// TIA Portal V17 export
// export: Created 2025-07-01T09:58:33.5756793Z, ExportSetting WithDefaults, DisplayName Totally Integrated Automation Portal, DisplayVersion V17 Update 8, DisplayName TIA Portal Openness, DisplayVersion V17 Update 8, DisplayName TIA Portal Version Control Interface, DisplayVersion V17, DisplayName SINAMICS Startdrive Advanced, DisplayVersion V17 SP2, DisplayName SINAMICS Startdrive G110M, G120, G120C, G120D, G120P, G115D, DisplayVersion V17 SP2, DisplayName SINAMICS Startdrive G130, G150, S120, S150, SINAMICS MV, S210, DisplayVersion V17 SP2, DisplayName STEP 7 Professional, DisplayVersion V17 Update 8, DisplayName SINUMERIK ONE STEP 7 Toolbox, DisplayVersion V17 Update 12, DisplayName SINUMERIK ONE PLC Basic Program Plus, DisplayVersion V17 Update 12, DisplayName SINUMERIK 840D sl STEP 7 Toolbox, DisplayVersion V17 Update 12, DisplayName STEP 7 Safety, DisplayVersion V17 Update 6, DisplayName WinCC Advanced, DisplayVersion V17 Update 8
FUNCTION "FC349_NCK_M_CH2_UNIT_1_STA_3" : Void   // FC349, LAD
TITLE = Channel 1 data
{ S7_Optimized_Access := 'FALSE' }
AUTHOR : ETXETAR
VERSION : 1.0
// stored: AutoNumber false, IsIECCheckEnabled false, SetENOAutomatically false, UDAEnableTagReadback false
BEGIN

REGION Network 1: ACKNOWLEDGE M704-FIXTURE 4 VERIFY PART AND TOOL IS CLAMPED DURING MACHINING (WHEN TRUE DO). TOGGLED / ACKNOWLEDGE M46-VERIFY FIXTURE 1 PART AND TOOL IS CLAMPED DURING
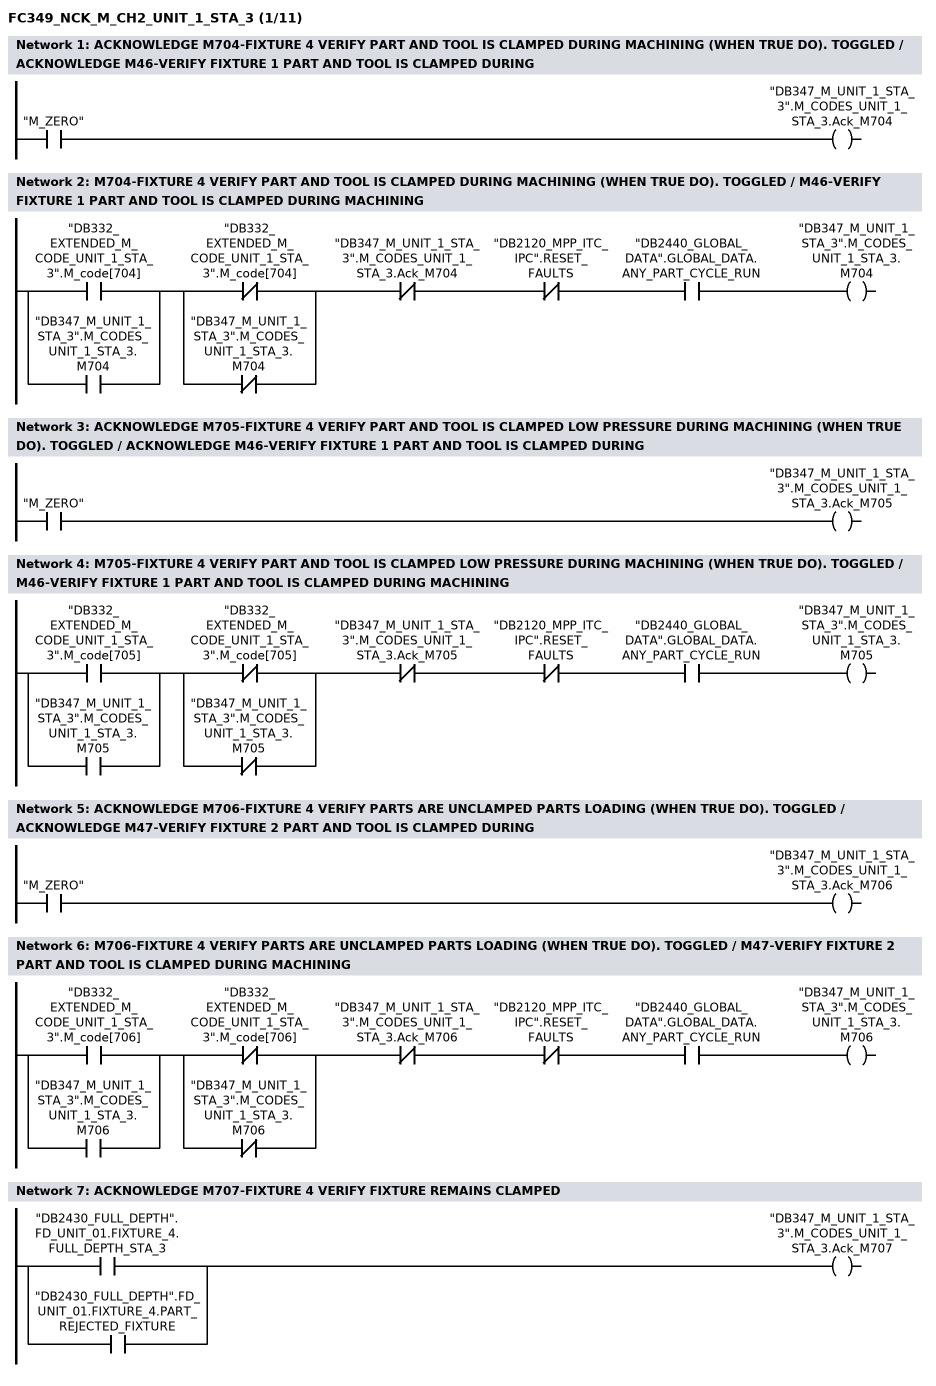
   RUNG wire#powerrail
      Contact( "M_ZERO" )
      Coil( "DB347_M_UNIT_1_STA_3".M_CODES_UNIT_1_STA_3.Ack_M704 )
   END_RUNG
   // the same network as SCL:
   "DB347_M_UNIT_1_STA_3".M_CODES_UNIT_1_STA_3.Ack_M704 := "M_ZERO";
END_REGION

REGION Network 2: M704-FIXTURE 4 VERIFY PART AND TOOL IS CLAMPED DURING MACHINING (WHEN TRUE DO). TOGGLED / M46-VERIFY FIXTURE 1 PART AND TOOL IS CLAMPED DURING MACHINING
   RUNG wire#powerrail
      Contact( "DB332_EXTENDED_M_CODE_UNIT_1_STA_3".M_code[704] )
      wire#w1
      I_Contact( "DB332_EXTENDED_M_CODE_UNIT_1_STA_3".M_code[704] )
      wire#w2
      I_Contact( "DB347_M_UNIT_1_STA_3".M_CODES_UNIT_1_STA_3.Ack_M704 )
      I_Contact( "DB2120_MPP_ITC_IPC".RESET_FAULTS )
      Contact( "DB2440_GLOBAL_DATA".GLOBAL_DATA.ANY_PART_CYCLE_RUN )
      Coil( "DB347_M_UNIT_1_STA_3".M_CODES_UNIT_1_STA_3.M704 )
   END_RUNG
   RUNG wire#powerrail
      Contact( "DB347_M_UNIT_1_STA_3".M_CODES_UNIT_1_STA_3.M704 )
   END_RUNG wire#w1
   RUNG wire#w1
      I_Contact( "DB347_M_UNIT_1_STA_3".M_CODES_UNIT_1_STA_3.M704 )
   END_RUNG wire#w2
   // the same network as SCL:
   "DB347_M_UNIT_1_STA_3".M_CODES_UNIT_1_STA_3.M704 := ("DB332_EXTENDED_M_CODE_UNIT_1_STA_3".M_code[704] OR "DB347_M_UNIT_1_STA_3".M_CODES_UNIT_1_STA_3.M704) AND (NOT "DB332_EXTENDED_M_CODE_UNIT_1_STA_3".M_code[704] OR NOT "DB347_M_UNIT_1_STA_3".M_CODES_UNIT_1_STA_3.M704) AND NOT "DB347_M_UNIT_1_STA_3".M_CODES_UNIT_1_STA_3.Ack_M704 AND NOT "DB2120_MPP_ITC_IPC".RESET_FAULTS AND "DB2440_GLOBAL_DATA".GLOBAL_DATA.ANY_PART_CYCLE_RUN;
END_REGION

REGION Network 3: ACKNOWLEDGE M705-FIXTURE 4 VERIFY PART AND TOOL IS CLAMPED LOW PRESSURE DURING MACHINING (WHEN TRUE DO). TOGGLED / ACKNOWLEDGE M46-VERIFY FIXTURE 1 PART AND TOOL IS CLAMPED DURING
   RUNG wire#powerrail
      Contact( "M_ZERO" )
      Coil( "DB347_M_UNIT_1_STA_3".M_CODES_UNIT_1_STA_3.Ack_M705 )
   END_RUNG
   // the same network as SCL:
   "DB347_M_UNIT_1_STA_3".M_CODES_UNIT_1_STA_3.Ack_M705 := "M_ZERO";
END_REGION

REGION Network 4: M705-FIXTURE 4 VERIFY PART AND TOOL IS CLAMPED LOW PRESSURE DURING MACHINING (WHEN TRUE DO). TOGGLED / M46-VERIFY FIXTURE 1 PART AND TOOL IS CLAMPED DURING MACHINING
   RUNG wire#powerrail
      Contact( "DB332_EXTENDED_M_CODE_UNIT_1_STA_3".M_code[705] )
      wire#w1
      I_Contact( "DB332_EXTENDED_M_CODE_UNIT_1_STA_3".M_code[705] )
      wire#w2
      I_Contact( "DB347_M_UNIT_1_STA_3".M_CODES_UNIT_1_STA_3.Ack_M705 )
      I_Contact( "DB2120_MPP_ITC_IPC".RESET_FAULTS )
      Contact( "DB2440_GLOBAL_DATA".GLOBAL_DATA.ANY_PART_CYCLE_RUN )
      Coil( "DB347_M_UNIT_1_STA_3".M_CODES_UNIT_1_STA_3.M705 )
   END_RUNG
   RUNG wire#powerrail
      Contact( "DB347_M_UNIT_1_STA_3".M_CODES_UNIT_1_STA_3.M705 )
   END_RUNG wire#w1
   RUNG wire#w1
      I_Contact( "DB347_M_UNIT_1_STA_3".M_CODES_UNIT_1_STA_3.M705 )
   END_RUNG wire#w2
   // the same network as SCL:
   "DB347_M_UNIT_1_STA_3".M_CODES_UNIT_1_STA_3.M705 := ("DB332_EXTENDED_M_CODE_UNIT_1_STA_3".M_code[705] OR "DB347_M_UNIT_1_STA_3".M_CODES_UNIT_1_STA_3.M705) AND (NOT "DB332_EXTENDED_M_CODE_UNIT_1_STA_3".M_code[705] OR NOT "DB347_M_UNIT_1_STA_3".M_CODES_UNIT_1_STA_3.M705) AND NOT "DB347_M_UNIT_1_STA_3".M_CODES_UNIT_1_STA_3.Ack_M705 AND NOT "DB2120_MPP_ITC_IPC".RESET_FAULTS AND "DB2440_GLOBAL_DATA".GLOBAL_DATA.ANY_PART_CYCLE_RUN;
END_REGION

REGION Network 5: ACKNOWLEDGE M706-FIXTURE 4 VERIFY PARTS ARE UNCLAMPED PARTS LOADING (WHEN TRUE DO). TOGGLED / ACKNOWLEDGE M47-VERIFY FIXTURE 2 PART AND TOOL IS CLAMPED DURING
   RUNG wire#powerrail
      Contact( "M_ZERO" )
      Coil( "DB347_M_UNIT_1_STA_3".M_CODES_UNIT_1_STA_3.Ack_M706 )
   END_RUNG
   // the same network as SCL:
   "DB347_M_UNIT_1_STA_3".M_CODES_UNIT_1_STA_3.Ack_M706 := "M_ZERO";
END_REGION

REGION Network 6: M706-FIXTURE 4 VERIFY PARTS ARE UNCLAMPED PARTS LOADING (WHEN TRUE DO). TOGGLED / M47-VERIFY FIXTURE 2 PART AND TOOL IS CLAMPED DURING MACHINING
   RUNG wire#powerrail
      Contact( "DB332_EXTENDED_M_CODE_UNIT_1_STA_3".M_code[706] )
      wire#w1
      I_Contact( "DB332_EXTENDED_M_CODE_UNIT_1_STA_3".M_code[706] )
      wire#w2
      I_Contact( "DB347_M_UNIT_1_STA_3".M_CODES_UNIT_1_STA_3.Ack_M706 )
      I_Contact( "DB2120_MPP_ITC_IPC".RESET_FAULTS )
      Contact( "DB2440_GLOBAL_DATA".GLOBAL_DATA.ANY_PART_CYCLE_RUN )
      Coil( "DB347_M_UNIT_1_STA_3".M_CODES_UNIT_1_STA_3.M706 )
   END_RUNG
   RUNG wire#powerrail
      Contact( "DB347_M_UNIT_1_STA_3".M_CODES_UNIT_1_STA_3.M706 )
   END_RUNG wire#w1
   RUNG wire#w1
      I_Contact( "DB347_M_UNIT_1_STA_3".M_CODES_UNIT_1_STA_3.M706 )
   END_RUNG wire#w2
   // the same network as SCL:
   "DB347_M_UNIT_1_STA_3".M_CODES_UNIT_1_STA_3.M706 := ("DB332_EXTENDED_M_CODE_UNIT_1_STA_3".M_code[706] OR "DB347_M_UNIT_1_STA_3".M_CODES_UNIT_1_STA_3.M706) AND (NOT "DB332_EXTENDED_M_CODE_UNIT_1_STA_3".M_code[706] OR NOT "DB347_M_UNIT_1_STA_3".M_CODES_UNIT_1_STA_3.M706) AND NOT "DB347_M_UNIT_1_STA_3".M_CODES_UNIT_1_STA_3.Ack_M706 AND NOT "DB2120_MPP_ITC_IPC".RESET_FAULTS AND "DB2440_GLOBAL_DATA".GLOBAL_DATA.ANY_PART_CYCLE_RUN;
END_REGION

REGION Network 7: ACKNOWLEDGE M707-FIXTURE 4 VERIFY FIXTURE REMAINS CLAMPED
   RUNG wire#powerrail
      Contact( "DB2430_FULL_DEPTH".FD_UNIT_01.FIXTURE_4.FULL_DEPTH_STA_3 )
      wire#w1
      Coil( "DB347_M_UNIT_1_STA_3".M_CODES_UNIT_1_STA_3.Ack_M707 )
   END_RUNG
   RUNG wire#powerrail
      Contact( "DB2430_FULL_DEPTH".FD_UNIT_01.FIXTURE_4.PART_REJECTED_FIXTURE )
   END_RUNG wire#w1
   // the same network as SCL:
   "DB347_M_UNIT_1_STA_3".M_CODES_UNIT_1_STA_3.Ack_M707 := "DB2430_FULL_DEPTH".FD_UNIT_01.FIXTURE_4.FULL_DEPTH_STA_3 OR "DB2430_FULL_DEPTH".FD_UNIT_01.FIXTURE_4.PART_REJECTED_FIXTURE;
END_REGION

REGION Network 8: M707-FIXTURE 4 VERIFY FIXTURE REMAINS CLAMPED
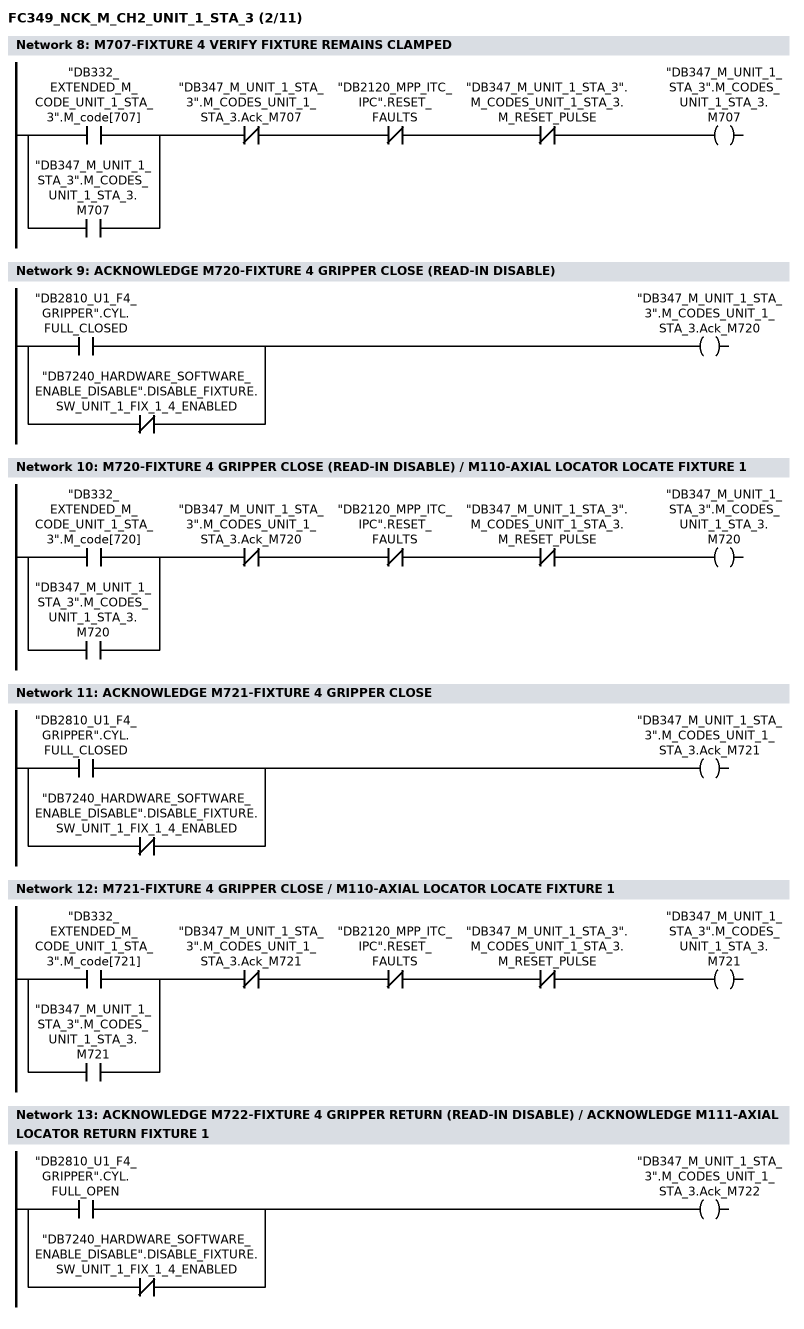
   RUNG wire#powerrail
      Contact( "DB332_EXTENDED_M_CODE_UNIT_1_STA_3".M_code[707] )
      wire#w1
      I_Contact( "DB347_M_UNIT_1_STA_3".M_CODES_UNIT_1_STA_3.Ack_M707 )
      I_Contact( "DB2120_MPP_ITC_IPC".RESET_FAULTS )
      I_Contact( "DB347_M_UNIT_1_STA_3".M_CODES_UNIT_1_STA_3.M_RESET_PULSE )
      Coil( "DB347_M_UNIT_1_STA_3".M_CODES_UNIT_1_STA_3.M707 )
   END_RUNG
   RUNG wire#powerrail
      Contact( "DB347_M_UNIT_1_STA_3".M_CODES_UNIT_1_STA_3.M707 )
   END_RUNG wire#w1
   // the same network as SCL:
   "DB347_M_UNIT_1_STA_3".M_CODES_UNIT_1_STA_3.M707 := ("DB332_EXTENDED_M_CODE_UNIT_1_STA_3".M_code[707] OR "DB347_M_UNIT_1_STA_3".M_CODES_UNIT_1_STA_3.M707) AND NOT "DB347_M_UNIT_1_STA_3".M_CODES_UNIT_1_STA_3.Ack_M707 AND NOT "DB2120_MPP_ITC_IPC".RESET_FAULTS AND NOT "DB347_M_UNIT_1_STA_3".M_CODES_UNIT_1_STA_3.M_RESET_PULSE;
END_REGION

REGION Network 9: ACKNOWLEDGE M720-FIXTURE 4 GRIPPER CLOSE (READ-IN DISABLE)
   RUNG wire#powerrail
      Contact( "DB2810_U1_F4_GRIPPER".CYL.FULL_CLOSED )
      wire#w1
      Coil( "DB347_M_UNIT_1_STA_3".M_CODES_UNIT_1_STA_3.Ack_M720 )
   END_RUNG
   RUNG wire#powerrail
      I_Contact( "DB7240_HARDWARE_SOFTWARE_ENABLE_DISABLE".DISABLE_FIXTURE.SW_UNIT_1_FIX_1_4_ENABLED )
   END_RUNG wire#w1
   // the same network as SCL:
   "DB347_M_UNIT_1_STA_3".M_CODES_UNIT_1_STA_3.Ack_M720 := "DB2810_U1_F4_GRIPPER".CYL.FULL_CLOSED OR NOT "DB7240_HARDWARE_SOFTWARE_ENABLE_DISABLE".DISABLE_FIXTURE.SW_UNIT_1_FIX_1_4_ENABLED;
END_REGION

REGION Network 10: M720-FIXTURE 4 GRIPPER CLOSE (READ-IN DISABLE) / M110-AXIAL LOCATOR LOCATE FIXTURE 1
   RUNG wire#powerrail
      Contact( "DB332_EXTENDED_M_CODE_UNIT_1_STA_3".M_code[720] )
      wire#w1
      I_Contact( "DB347_M_UNIT_1_STA_3".M_CODES_UNIT_1_STA_3.Ack_M720 )
      I_Contact( "DB2120_MPP_ITC_IPC".RESET_FAULTS )
      I_Contact( "DB347_M_UNIT_1_STA_3".M_CODES_UNIT_1_STA_3.M_RESET_PULSE )
      Coil( "DB347_M_UNIT_1_STA_3".M_CODES_UNIT_1_STA_3.M720 )
   END_RUNG
   RUNG wire#powerrail
      Contact( "DB347_M_UNIT_1_STA_3".M_CODES_UNIT_1_STA_3.M720 )
   END_RUNG wire#w1
   // the same network as SCL:
   "DB347_M_UNIT_1_STA_3".M_CODES_UNIT_1_STA_3.M720 := ("DB332_EXTENDED_M_CODE_UNIT_1_STA_3".M_code[720] OR "DB347_M_UNIT_1_STA_3".M_CODES_UNIT_1_STA_3.M720) AND NOT "DB347_M_UNIT_1_STA_3".M_CODES_UNIT_1_STA_3.Ack_M720 AND NOT "DB2120_MPP_ITC_IPC".RESET_FAULTS AND NOT "DB347_M_UNIT_1_STA_3".M_CODES_UNIT_1_STA_3.M_RESET_PULSE;
END_REGION

REGION Network 11: ACKNOWLEDGE M721-FIXTURE 4 GRIPPER CLOSE
   RUNG wire#powerrail
      Contact( "DB2810_U1_F4_GRIPPER".CYL.FULL_CLOSED )
      wire#w1
      Coil( "DB347_M_UNIT_1_STA_3".M_CODES_UNIT_1_STA_3.Ack_M721 )
   END_RUNG
   RUNG wire#powerrail
      I_Contact( "DB7240_HARDWARE_SOFTWARE_ENABLE_DISABLE".DISABLE_FIXTURE.SW_UNIT_1_FIX_1_4_ENABLED )
   END_RUNG wire#w1
   // the same network as SCL:
   "DB347_M_UNIT_1_STA_3".M_CODES_UNIT_1_STA_3.Ack_M721 := "DB2810_U1_F4_GRIPPER".CYL.FULL_CLOSED OR NOT "DB7240_HARDWARE_SOFTWARE_ENABLE_DISABLE".DISABLE_FIXTURE.SW_UNIT_1_FIX_1_4_ENABLED;
END_REGION

REGION Network 12: M721-FIXTURE 4 GRIPPER CLOSE / M110-AXIAL LOCATOR LOCATE FIXTURE 1
   RUNG wire#powerrail
      Contact( "DB332_EXTENDED_M_CODE_UNIT_1_STA_3".M_code[721] )
      wire#w1
      I_Contact( "DB347_M_UNIT_1_STA_3".M_CODES_UNIT_1_STA_3.Ack_M721 )
      I_Contact( "DB2120_MPP_ITC_IPC".RESET_FAULTS )
      I_Contact( "DB347_M_UNIT_1_STA_3".M_CODES_UNIT_1_STA_3.M_RESET_PULSE )
      Coil( "DB347_M_UNIT_1_STA_3".M_CODES_UNIT_1_STA_3.M721 )
   END_RUNG
   RUNG wire#powerrail
      Contact( "DB347_M_UNIT_1_STA_3".M_CODES_UNIT_1_STA_3.M721 )
   END_RUNG wire#w1
   // the same network as SCL:
   "DB347_M_UNIT_1_STA_3".M_CODES_UNIT_1_STA_3.M721 := ("DB332_EXTENDED_M_CODE_UNIT_1_STA_3".M_code[721] OR "DB347_M_UNIT_1_STA_3".M_CODES_UNIT_1_STA_3.M721) AND NOT "DB347_M_UNIT_1_STA_3".M_CODES_UNIT_1_STA_3.Ack_M721 AND NOT "DB2120_MPP_ITC_IPC".RESET_FAULTS AND NOT "DB347_M_UNIT_1_STA_3".M_CODES_UNIT_1_STA_3.M_RESET_PULSE;
END_REGION

REGION Network 13: ACKNOWLEDGE M722-FIXTURE 4 GRIPPER RETURN (READ-IN DISABLE) / ACKNOWLEDGE M111-AXIAL LOCATOR RETURN FIXTURE 1
   RUNG wire#powerrail
      Contact( "DB2810_U1_F4_GRIPPER".CYL.FULL_OPEN )
      wire#w1
      Coil( "DB347_M_UNIT_1_STA_3".M_CODES_UNIT_1_STA_3.Ack_M722 )
   END_RUNG
   RUNG wire#powerrail
      I_Contact( "DB7240_HARDWARE_SOFTWARE_ENABLE_DISABLE".DISABLE_FIXTURE.SW_UNIT_1_FIX_1_4_ENABLED )
   END_RUNG wire#w1
   // the same network as SCL:
   "DB347_M_UNIT_1_STA_3".M_CODES_UNIT_1_STA_3.Ack_M722 := "DB2810_U1_F4_GRIPPER".CYL.FULL_OPEN OR NOT "DB7240_HARDWARE_SOFTWARE_ENABLE_DISABLE".DISABLE_FIXTURE.SW_UNIT_1_FIX_1_4_ENABLED;
END_REGION

REGION Network 14: M722-FIXTURE 4 GRIPPER RETURN (READ-IN DISABLE) / M111-AXIAL LOCATOR RETURN FIXTURE 1
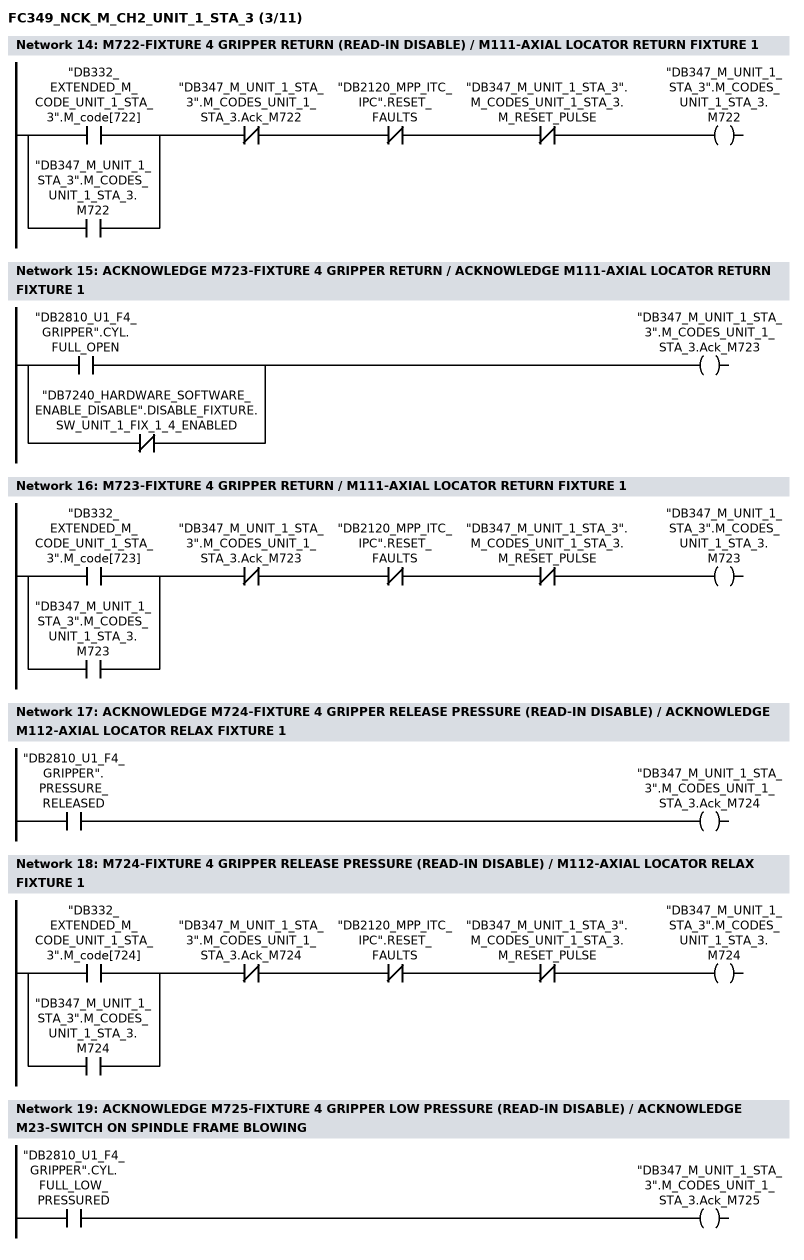
   RUNG wire#powerrail
      Contact( "DB332_EXTENDED_M_CODE_UNIT_1_STA_3".M_code[722] )
      wire#w1
      I_Contact( "DB347_M_UNIT_1_STA_3".M_CODES_UNIT_1_STA_3.Ack_M722 )
      I_Contact( "DB2120_MPP_ITC_IPC".RESET_FAULTS )
      I_Contact( "DB347_M_UNIT_1_STA_3".M_CODES_UNIT_1_STA_3.M_RESET_PULSE )
      Coil( "DB347_M_UNIT_1_STA_3".M_CODES_UNIT_1_STA_3.M722 )
   END_RUNG
   RUNG wire#powerrail
      Contact( "DB347_M_UNIT_1_STA_3".M_CODES_UNIT_1_STA_3.M722 )
   END_RUNG wire#w1
   // the same network as SCL:
   "DB347_M_UNIT_1_STA_3".M_CODES_UNIT_1_STA_3.M722 := ("DB332_EXTENDED_M_CODE_UNIT_1_STA_3".M_code[722] OR "DB347_M_UNIT_1_STA_3".M_CODES_UNIT_1_STA_3.M722) AND NOT "DB347_M_UNIT_1_STA_3".M_CODES_UNIT_1_STA_3.Ack_M722 AND NOT "DB2120_MPP_ITC_IPC".RESET_FAULTS AND NOT "DB347_M_UNIT_1_STA_3".M_CODES_UNIT_1_STA_3.M_RESET_PULSE;
END_REGION

REGION Network 15: ACKNOWLEDGE M723-FIXTURE 4 GRIPPER RETURN / ACKNOWLEDGE M111-AXIAL LOCATOR RETURN FIXTURE 1
   RUNG wire#powerrail
      Contact( "DB2810_U1_F4_GRIPPER".CYL.FULL_OPEN )
      wire#w1
      Coil( "DB347_M_UNIT_1_STA_3".M_CODES_UNIT_1_STA_3.Ack_M723 )
   END_RUNG
   RUNG wire#powerrail
      I_Contact( "DB7240_HARDWARE_SOFTWARE_ENABLE_DISABLE".DISABLE_FIXTURE.SW_UNIT_1_FIX_1_4_ENABLED )
   END_RUNG wire#w1
   // the same network as SCL:
   "DB347_M_UNIT_1_STA_3".M_CODES_UNIT_1_STA_3.Ack_M723 := "DB2810_U1_F4_GRIPPER".CYL.FULL_OPEN OR NOT "DB7240_HARDWARE_SOFTWARE_ENABLE_DISABLE".DISABLE_FIXTURE.SW_UNIT_1_FIX_1_4_ENABLED;
END_REGION

REGION Network 16: M723-FIXTURE 4 GRIPPER RETURN / M111-AXIAL LOCATOR RETURN FIXTURE 1
   RUNG wire#powerrail
      Contact( "DB332_EXTENDED_M_CODE_UNIT_1_STA_3".M_code[723] )
      wire#w1
      I_Contact( "DB347_M_UNIT_1_STA_3".M_CODES_UNIT_1_STA_3.Ack_M723 )
      I_Contact( "DB2120_MPP_ITC_IPC".RESET_FAULTS )
      I_Contact( "DB347_M_UNIT_1_STA_3".M_CODES_UNIT_1_STA_3.M_RESET_PULSE )
      Coil( "DB347_M_UNIT_1_STA_3".M_CODES_UNIT_1_STA_3.M723 )
   END_RUNG
   RUNG wire#powerrail
      Contact( "DB347_M_UNIT_1_STA_3".M_CODES_UNIT_1_STA_3.M723 )
   END_RUNG wire#w1
   // the same network as SCL:
   "DB347_M_UNIT_1_STA_3".M_CODES_UNIT_1_STA_3.M723 := ("DB332_EXTENDED_M_CODE_UNIT_1_STA_3".M_code[723] OR "DB347_M_UNIT_1_STA_3".M_CODES_UNIT_1_STA_3.M723) AND NOT "DB347_M_UNIT_1_STA_3".M_CODES_UNIT_1_STA_3.Ack_M723 AND NOT "DB2120_MPP_ITC_IPC".RESET_FAULTS AND NOT "DB347_M_UNIT_1_STA_3".M_CODES_UNIT_1_STA_3.M_RESET_PULSE;
END_REGION

REGION Network 17: ACKNOWLEDGE M724-FIXTURE 4 GRIPPER RELEASE PRESSURE (READ-IN DISABLE) / ACKNOWLEDGE M112-AXIAL LOCATOR RELAX FIXTURE 1
   RUNG wire#powerrail
      Contact( "DB2810_U1_F4_GRIPPER".PRESSURE_RELEASED )
      Coil( "DB347_M_UNIT_1_STA_3".M_CODES_UNIT_1_STA_3.Ack_M724 )
   END_RUNG
   // the same network as SCL:
   "DB347_M_UNIT_1_STA_3".M_CODES_UNIT_1_STA_3.Ack_M724 := "DB2810_U1_F4_GRIPPER".PRESSURE_RELEASED;
END_REGION

REGION Network 18: M724-FIXTURE 4 GRIPPER RELEASE PRESSURE (READ-IN DISABLE) / M112-AXIAL LOCATOR RELAX FIXTURE 1
   RUNG wire#powerrail
      Contact( "DB332_EXTENDED_M_CODE_UNIT_1_STA_3".M_code[724] )
      wire#w1
      I_Contact( "DB347_M_UNIT_1_STA_3".M_CODES_UNIT_1_STA_3.Ack_M724 )
      I_Contact( "DB2120_MPP_ITC_IPC".RESET_FAULTS )
      I_Contact( "DB347_M_UNIT_1_STA_3".M_CODES_UNIT_1_STA_3.M_RESET_PULSE )
      Coil( "DB347_M_UNIT_1_STA_3".M_CODES_UNIT_1_STA_3.M724 )
   END_RUNG
   RUNG wire#powerrail
      Contact( "DB347_M_UNIT_1_STA_3".M_CODES_UNIT_1_STA_3.M724 )
   END_RUNG wire#w1
   // the same network as SCL:
   "DB347_M_UNIT_1_STA_3".M_CODES_UNIT_1_STA_3.M724 := ("DB332_EXTENDED_M_CODE_UNIT_1_STA_3".M_code[724] OR "DB347_M_UNIT_1_STA_3".M_CODES_UNIT_1_STA_3.M724) AND NOT "DB347_M_UNIT_1_STA_3".M_CODES_UNIT_1_STA_3.Ack_M724 AND NOT "DB2120_MPP_ITC_IPC".RESET_FAULTS AND NOT "DB347_M_UNIT_1_STA_3".M_CODES_UNIT_1_STA_3.M_RESET_PULSE;
END_REGION

REGION Network 19: ACKNOWLEDGE M725-FIXTURE 4 GRIPPER LOW PRESSURE (READ-IN DISABLE) / ACKNOWLEDGE M23-SWITCH ON SPINDLE FRAME BLOWING
   RUNG wire#powerrail
      Contact( "DB2810_U1_F4_GRIPPER".CYL.FULL_LOW_PRESSURED )
      Coil( "DB347_M_UNIT_1_STA_3".M_CODES_UNIT_1_STA_3.Ack_M725 )
   END_RUNG
   // the same network as SCL:
   "DB347_M_UNIT_1_STA_3".M_CODES_UNIT_1_STA_3.Ack_M725 := "DB2810_U1_F4_GRIPPER".CYL.FULL_LOW_PRESSURED;
END_REGION

REGION Network 20: M725-FIXTURE 4 GRIPPER LOW PRESSURE (READ-IN DISABLE) / M23-SWITCH ON SPINDLE FRAME BLOWING
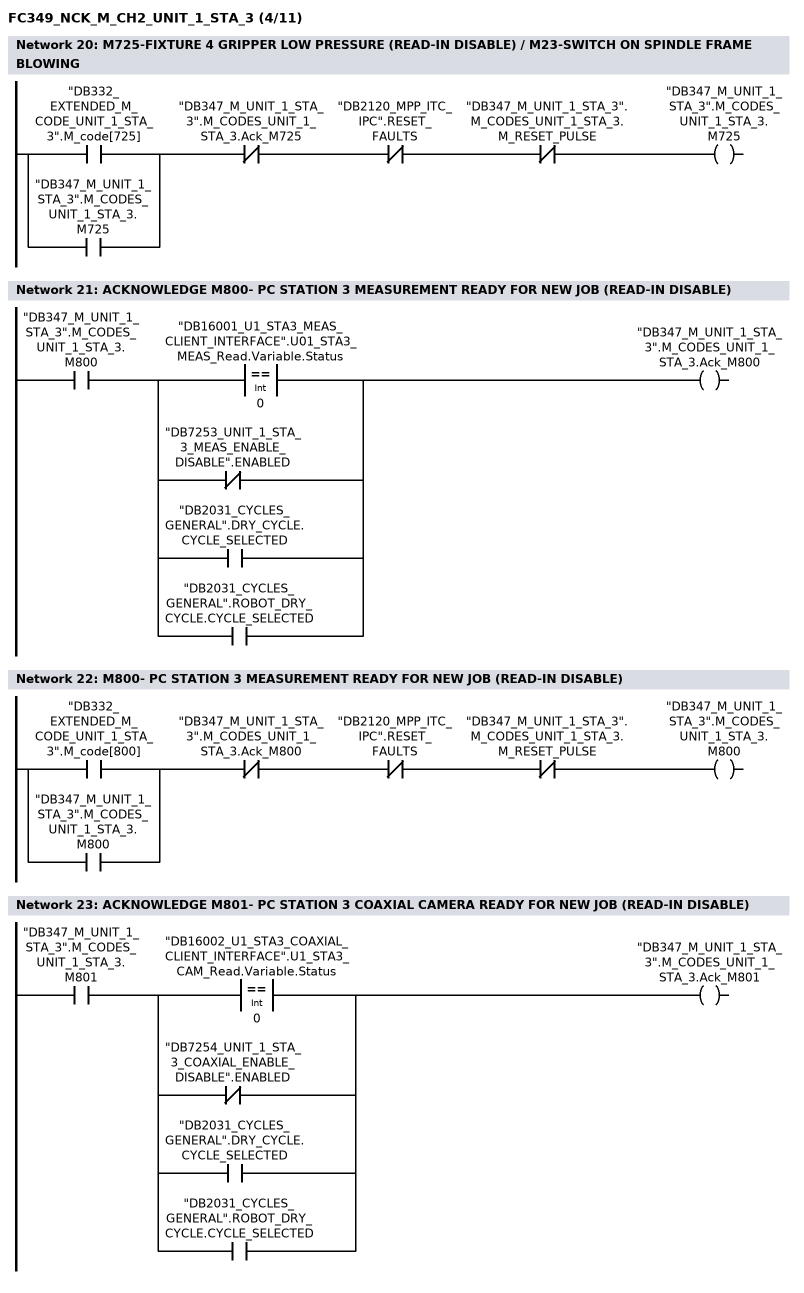
   RUNG wire#powerrail
      Contact( "DB332_EXTENDED_M_CODE_UNIT_1_STA_3".M_code[725] )
      wire#w1
      I_Contact( "DB347_M_UNIT_1_STA_3".M_CODES_UNIT_1_STA_3.Ack_M725 )
      I_Contact( "DB2120_MPP_ITC_IPC".RESET_FAULTS )
      I_Contact( "DB347_M_UNIT_1_STA_3".M_CODES_UNIT_1_STA_3.M_RESET_PULSE )
      Coil( "DB347_M_UNIT_1_STA_3".M_CODES_UNIT_1_STA_3.M725 )
   END_RUNG
   RUNG wire#powerrail
      Contact( "DB347_M_UNIT_1_STA_3".M_CODES_UNIT_1_STA_3.M725 )
   END_RUNG wire#w1
   // the same network as SCL:
   "DB347_M_UNIT_1_STA_3".M_CODES_UNIT_1_STA_3.M725 := ("DB332_EXTENDED_M_CODE_UNIT_1_STA_3".M_code[725] OR "DB347_M_UNIT_1_STA_3".M_CODES_UNIT_1_STA_3.M725) AND NOT "DB347_M_UNIT_1_STA_3".M_CODES_UNIT_1_STA_3.Ack_M725 AND NOT "DB2120_MPP_ITC_IPC".RESET_FAULTS AND NOT "DB347_M_UNIT_1_STA_3".M_CODES_UNIT_1_STA_3.M_RESET_PULSE;
END_REGION

REGION Network 21: ACKNOWLEDGE M800- PC STATION 3 MEASUREMENT READY FOR NEW JOB (READ-IN DISABLE)
   RUNG wire#powerrail
      Contact( "DB347_M_UNIT_1_STA_3".M_CODES_UNIT_1_STA_3.M800 )
      wire#w1
      { S7_Templates := "SrcType := Int" } EQ_Contact(in1 := "DB16001_U1_STA3_MEAS_CLIENT_INTERFACE".U01_STA3_MEAS_Read.Variable.Status, in2 := 0)
      wire#w2
      Coil( "DB347_M_UNIT_1_STA_3".M_CODES_UNIT_1_STA_3.Ack_M800 )
   END_RUNG
   RUNG wire#w1
      I_Contact( "DB7253_UNIT_1_STA_3_MEAS_ENABLE_DISABLE".ENABLED )
   END_RUNG wire#w2
   RUNG wire#w1
      Contact( "DB2031_CYCLES_GENERAL".DRY_CYCLE.CYCLE_SELECTED )
   END_RUNG wire#w2
   RUNG wire#w1
      Contact( "DB2031_CYCLES_GENERAL".ROBOT_DRY_CYCLE.CYCLE_SELECTED )
   END_RUNG wire#w2
   // the same network as SCL:
   "DB347_M_UNIT_1_STA_3".M_CODES_UNIT_1_STA_3.Ack_M800 := "DB347_M_UNIT_1_STA_3".M_CODES_UNIT_1_STA_3.M800 AND (("DB16001_U1_STA3_MEAS_CLIENT_INTERFACE".U01_STA3_MEAS_Read.Variable.Status = 0) OR NOT "DB7253_UNIT_1_STA_3_MEAS_ENABLE_DISABLE".ENABLED OR "DB2031_CYCLES_GENERAL".DRY_CYCLE.CYCLE_SELECTED OR "DB2031_CYCLES_GENERAL".ROBOT_DRY_CYCLE.CYCLE_SELECTED);
END_REGION

REGION Network 22: M800- PC STATION 3 MEASUREMENT READY FOR NEW JOB (READ-IN DISABLE)
   RUNG wire#powerrail
      Contact( "DB332_EXTENDED_M_CODE_UNIT_1_STA_3".M_code[800] )
      wire#w1
      I_Contact( "DB347_M_UNIT_1_STA_3".M_CODES_UNIT_1_STA_3.Ack_M800 )
      I_Contact( "DB2120_MPP_ITC_IPC".RESET_FAULTS )
      I_Contact( "DB347_M_UNIT_1_STA_3".M_CODES_UNIT_1_STA_3.M_RESET_PULSE )
      Coil( "DB347_M_UNIT_1_STA_3".M_CODES_UNIT_1_STA_3.M800 )
   END_RUNG
   RUNG wire#powerrail
      Contact( "DB347_M_UNIT_1_STA_3".M_CODES_UNIT_1_STA_3.M800 )
   END_RUNG wire#w1
   // the same network as SCL:
   "DB347_M_UNIT_1_STA_3".M_CODES_UNIT_1_STA_3.M800 := ("DB332_EXTENDED_M_CODE_UNIT_1_STA_3".M_code[800] OR "DB347_M_UNIT_1_STA_3".M_CODES_UNIT_1_STA_3.M800) AND NOT "DB347_M_UNIT_1_STA_3".M_CODES_UNIT_1_STA_3.Ack_M800 AND NOT "DB2120_MPP_ITC_IPC".RESET_FAULTS AND NOT "DB347_M_UNIT_1_STA_3".M_CODES_UNIT_1_STA_3.M_RESET_PULSE;
END_REGION

REGION Network 23: ACKNOWLEDGE M801- PC STATION 3 COAXIAL CAMERA READY FOR NEW JOB (READ-IN DISABLE)
   RUNG wire#powerrail
      Contact( "DB347_M_UNIT_1_STA_3".M_CODES_UNIT_1_STA_3.M801 )
      wire#w1
      { S7_Templates := "SrcType := Int" } EQ_Contact(in1 := "DB16002_U1_STA3_COAXIAL_CLIENT_INTERFACE".U1_STA3_CAM_Read.Variable.Status, in2 := 0)
      wire#w2
      Coil( "DB347_M_UNIT_1_STA_3".M_CODES_UNIT_1_STA_3.Ack_M801 )
   END_RUNG
   RUNG wire#w1
      I_Contact( "DB7254_UNIT_1_STA_3_COAXIAL_ENABLE_DISABLE".ENABLED )
   END_RUNG wire#w2
   RUNG wire#w1
      Contact( "DB2031_CYCLES_GENERAL".DRY_CYCLE.CYCLE_SELECTED )
   END_RUNG wire#w2
   RUNG wire#w1
      Contact( "DB2031_CYCLES_GENERAL".ROBOT_DRY_CYCLE.CYCLE_SELECTED )
   END_RUNG wire#w2
   // the same network as SCL:
   "DB347_M_UNIT_1_STA_3".M_CODES_UNIT_1_STA_3.Ack_M801 := "DB347_M_UNIT_1_STA_3".M_CODES_UNIT_1_STA_3.M801 AND (("DB16002_U1_STA3_COAXIAL_CLIENT_INTERFACE".U1_STA3_CAM_Read.Variable.Status = 0) OR NOT "DB7254_UNIT_1_STA_3_COAXIAL_ENABLE_DISABLE".ENABLED OR "DB2031_CYCLES_GENERAL".DRY_CYCLE.CYCLE_SELECTED OR "DB2031_CYCLES_GENERAL".ROBOT_DRY_CYCLE.CYCLE_SELECTED);
END_REGION

REGION Network 24: M801- PC STATION 3 CAOXIAL CAMERA READY FOR NEW JOB (READ-IN DISABLE)
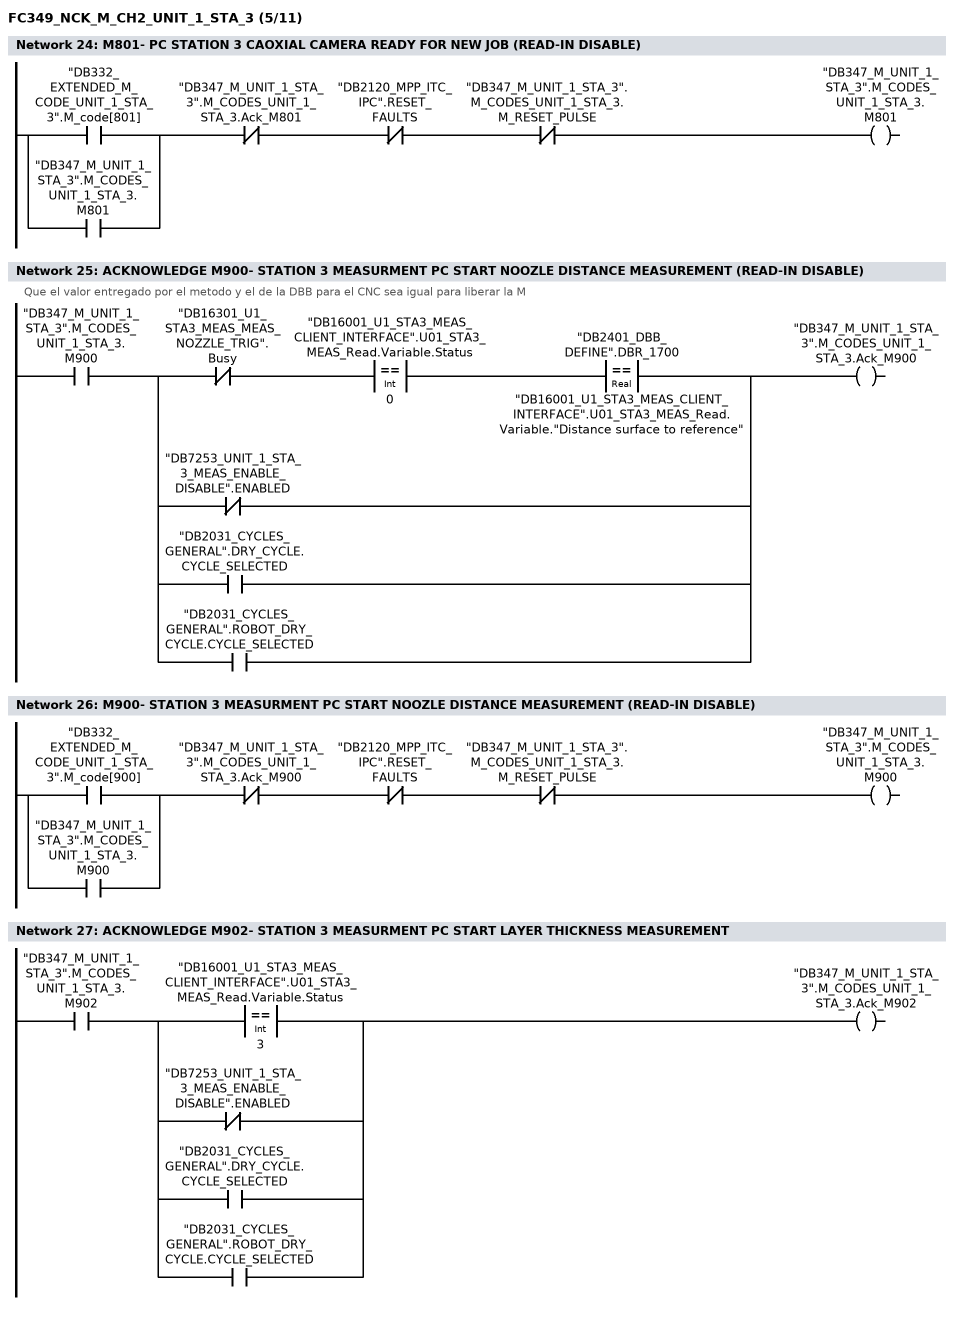
   RUNG wire#powerrail
      Contact( "DB332_EXTENDED_M_CODE_UNIT_1_STA_3".M_code[801] )
      wire#w1
      I_Contact( "DB347_M_UNIT_1_STA_3".M_CODES_UNIT_1_STA_3.Ack_M801 )
      I_Contact( "DB2120_MPP_ITC_IPC".RESET_FAULTS )
      I_Contact( "DB347_M_UNIT_1_STA_3".M_CODES_UNIT_1_STA_3.M_RESET_PULSE )
      Coil( "DB347_M_UNIT_1_STA_3".M_CODES_UNIT_1_STA_3.M801 )
   END_RUNG
   RUNG wire#powerrail
      Contact( "DB347_M_UNIT_1_STA_3".M_CODES_UNIT_1_STA_3.M801 )
   END_RUNG wire#w1
   // the same network as SCL:
   "DB347_M_UNIT_1_STA_3".M_CODES_UNIT_1_STA_3.M801 := ("DB332_EXTENDED_M_CODE_UNIT_1_STA_3".M_code[801] OR "DB347_M_UNIT_1_STA_3".M_CODES_UNIT_1_STA_3.M801) AND NOT "DB347_M_UNIT_1_STA_3".M_CODES_UNIT_1_STA_3.Ack_M801 AND NOT "DB2120_MPP_ITC_IPC".RESET_FAULTS AND NOT "DB347_M_UNIT_1_STA_3".M_CODES_UNIT_1_STA_3.M_RESET_PULSE;
END_REGION

REGION Network 25: ACKNOWLEDGE M900- STATION 3 MEASURMENT PC START NOOZLE DISTANCE MEASUREMENT (READ-IN DISABLE)
   // Que el valor entregado por el metodo y el de la DBB para el CNC sea igual para liberar la M
   RUNG wire#powerrail
      Contact( "DB347_M_UNIT_1_STA_3".M_CODES_UNIT_1_STA_3.M900 )
      wire#w1
      I_Contact( "DB16301_U1_STA3_MEAS_MEAS_NOZZLE_TRIG".Busy )
      { S7_Templates := "SrcType := Int" } EQ_Contact(in1 := "DB16001_U1_STA3_MEAS_CLIENT_INTERFACE".U01_STA3_MEAS_Read.Variable.Status, in2 := 0)
      { S7_Templates := "SrcType := Real" } EQ_Contact(in1 := "DB2401_DBB_DEFINE".DBR_1700, in2 := "DB16001_U1_STA3_MEAS_CLIENT_INTERFACE".U01_STA3_MEAS_Read.Variable."Distance surface to reference")
      wire#w2
      Coil( "DB347_M_UNIT_1_STA_3".M_CODES_UNIT_1_STA_3.Ack_M900 )
   END_RUNG
   RUNG wire#w1
      I_Contact( "DB7253_UNIT_1_STA_3_MEAS_ENABLE_DISABLE".ENABLED )
   END_RUNG wire#w2
   RUNG wire#w1
      Contact( "DB2031_CYCLES_GENERAL".DRY_CYCLE.CYCLE_SELECTED )
   END_RUNG wire#w2
   RUNG wire#w1
      Contact( "DB2031_CYCLES_GENERAL".ROBOT_DRY_CYCLE.CYCLE_SELECTED )
   END_RUNG wire#w2
   // the same network as SCL:
   "DB347_M_UNIT_1_STA_3".M_CODES_UNIT_1_STA_3.Ack_M900 := "DB347_M_UNIT_1_STA_3".M_CODES_UNIT_1_STA_3.M900 AND ((NOT "DB16301_U1_STA3_MEAS_MEAS_NOZZLE_TRIG".Busy AND ("DB16001_U1_STA3_MEAS_CLIENT_INTERFACE".U01_STA3_MEAS_Read.Variable.Status = 0) AND ("DB2401_DBB_DEFINE".DBR_1700 = "DB16001_U1_STA3_MEAS_CLIENT_INTERFACE".U01_STA3_MEAS_Read.Variable."Distance surface to reference")) OR NOT "DB7253_UNIT_1_STA_3_MEAS_ENABLE_DISABLE".ENABLED OR "DB2031_CYCLES_GENERAL".DRY_CYCLE.CYCLE_SELECTED OR "DB2031_CYCLES_GENERAL".ROBOT_DRY_CYCLE.CYCLE_SELECTED);
END_REGION

REGION Network 26: M900- STATION 3 MEASURMENT PC START NOOZLE DISTANCE MEASUREMENT (READ-IN DISABLE)
   RUNG wire#powerrail
      Contact( "DB332_EXTENDED_M_CODE_UNIT_1_STA_3".M_code[900] )
      wire#w1
      I_Contact( "DB347_M_UNIT_1_STA_3".M_CODES_UNIT_1_STA_3.Ack_M900 )
      I_Contact( "DB2120_MPP_ITC_IPC".RESET_FAULTS )
      I_Contact( "DB347_M_UNIT_1_STA_3".M_CODES_UNIT_1_STA_3.M_RESET_PULSE )
      Coil( "DB347_M_UNIT_1_STA_3".M_CODES_UNIT_1_STA_3.M900 )
   END_RUNG
   RUNG wire#powerrail
      Contact( "DB347_M_UNIT_1_STA_3".M_CODES_UNIT_1_STA_3.M900 )
   END_RUNG wire#w1
   // the same network as SCL:
   "DB347_M_UNIT_1_STA_3".M_CODES_UNIT_1_STA_3.M900 := ("DB332_EXTENDED_M_CODE_UNIT_1_STA_3".M_code[900] OR "DB347_M_UNIT_1_STA_3".M_CODES_UNIT_1_STA_3.M900) AND NOT "DB347_M_UNIT_1_STA_3".M_CODES_UNIT_1_STA_3.Ack_M900 AND NOT "DB2120_MPP_ITC_IPC".RESET_FAULTS AND NOT "DB347_M_UNIT_1_STA_3".M_CODES_UNIT_1_STA_3.M_RESET_PULSE;
END_REGION

REGION Network 27: ACKNOWLEDGE M902- STATION 3 MEASURMENT PC START LAYER THICKNESS MEASUREMENT
   RUNG wire#powerrail
      Contact( "DB347_M_UNIT_1_STA_3".M_CODES_UNIT_1_STA_3.M902 )
      wire#w1
      { S7_Templates := "SrcType := Int" } EQ_Contact(in1 := "DB16001_U1_STA3_MEAS_CLIENT_INTERFACE".U01_STA3_MEAS_Read.Variable.Status, in2 := 3)
      wire#w2
      Coil( "DB347_M_UNIT_1_STA_3".M_CODES_UNIT_1_STA_3.Ack_M902 )
   END_RUNG
   RUNG wire#w1
      I_Contact( "DB7253_UNIT_1_STA_3_MEAS_ENABLE_DISABLE".ENABLED )
   END_RUNG wire#w2
   RUNG wire#w1
      Contact( "DB2031_CYCLES_GENERAL".DRY_CYCLE.CYCLE_SELECTED )
   END_RUNG wire#w2
   RUNG wire#w1
      Contact( "DB2031_CYCLES_GENERAL".ROBOT_DRY_CYCLE.CYCLE_SELECTED )
   END_RUNG wire#w2
   // the same network as SCL:
   "DB347_M_UNIT_1_STA_3".M_CODES_UNIT_1_STA_3.Ack_M902 := "DB347_M_UNIT_1_STA_3".M_CODES_UNIT_1_STA_3.M902 AND (("DB16001_U1_STA3_MEAS_CLIENT_INTERFACE".U01_STA3_MEAS_Read.Variable.Status = 3) OR NOT "DB7253_UNIT_1_STA_3_MEAS_ENABLE_DISABLE".ENABLED OR "DB2031_CYCLES_GENERAL".DRY_CYCLE.CYCLE_SELECTED OR "DB2031_CYCLES_GENERAL".ROBOT_DRY_CYCLE.CYCLE_SELECTED);
END_REGION

REGION Network 28: M902- STATION 3 MEASURMENT PC START LAYER THICKNESS MEASUREMENT
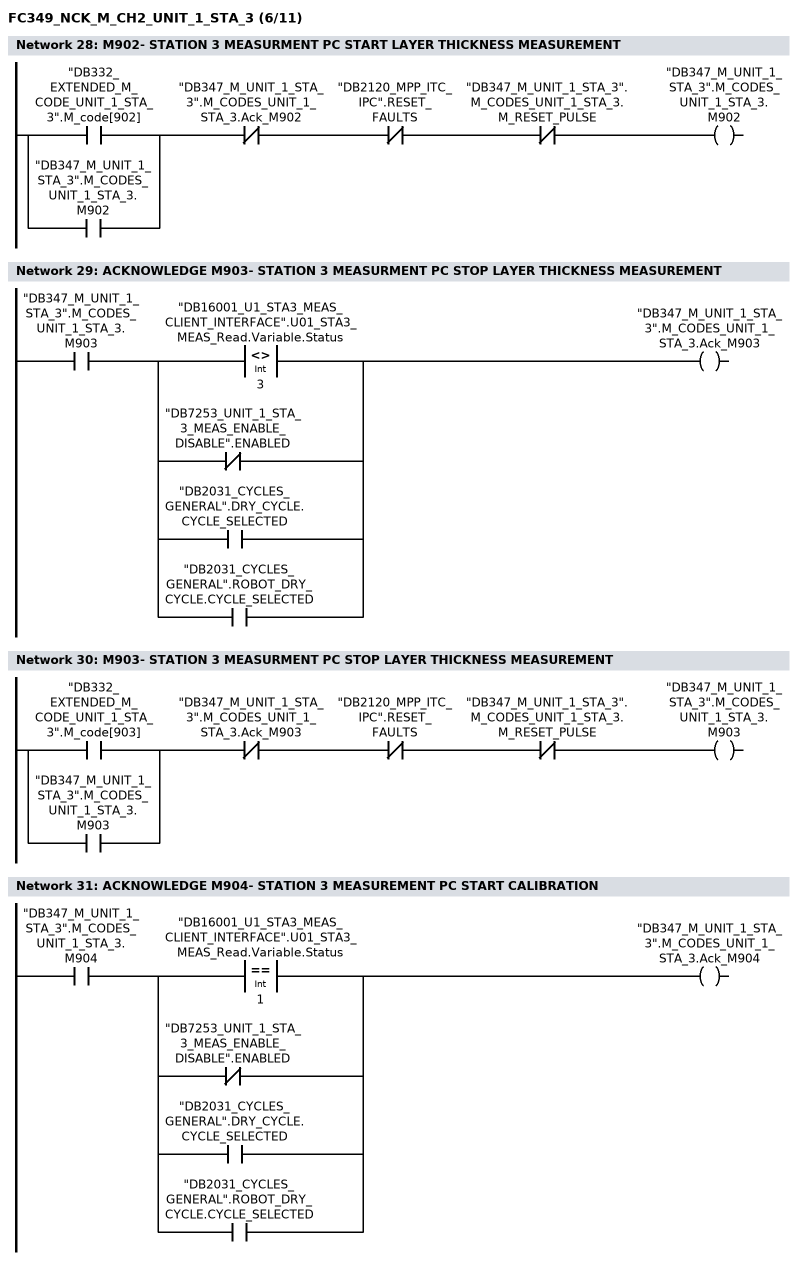
   RUNG wire#powerrail
      Contact( "DB332_EXTENDED_M_CODE_UNIT_1_STA_3".M_code[902] )
      wire#w1
      I_Contact( "DB347_M_UNIT_1_STA_3".M_CODES_UNIT_1_STA_3.Ack_M902 )
      I_Contact( "DB2120_MPP_ITC_IPC".RESET_FAULTS )
      I_Contact( "DB347_M_UNIT_1_STA_3".M_CODES_UNIT_1_STA_3.M_RESET_PULSE )
      Coil( "DB347_M_UNIT_1_STA_3".M_CODES_UNIT_1_STA_3.M902 )
   END_RUNG
   RUNG wire#powerrail
      Contact( "DB347_M_UNIT_1_STA_3".M_CODES_UNIT_1_STA_3.M902 )
   END_RUNG wire#w1
   // the same network as SCL:
   "DB347_M_UNIT_1_STA_3".M_CODES_UNIT_1_STA_3.M902 := ("DB332_EXTENDED_M_CODE_UNIT_1_STA_3".M_code[902] OR "DB347_M_UNIT_1_STA_3".M_CODES_UNIT_1_STA_3.M902) AND NOT "DB347_M_UNIT_1_STA_3".M_CODES_UNIT_1_STA_3.Ack_M902 AND NOT "DB2120_MPP_ITC_IPC".RESET_FAULTS AND NOT "DB347_M_UNIT_1_STA_3".M_CODES_UNIT_1_STA_3.M_RESET_PULSE;
END_REGION

REGION Network 29: ACKNOWLEDGE M903- STATION 3 MEASURMENT PC STOP LAYER THICKNESS MEASUREMENT
   RUNG wire#powerrail
      Contact( "DB347_M_UNIT_1_STA_3".M_CODES_UNIT_1_STA_3.M903 )
      wire#w1
      { S7_Templates := "SrcType := Int" } NE_Contact(in1 := "DB16001_U1_STA3_MEAS_CLIENT_INTERFACE".U01_STA3_MEAS_Read.Variable.Status, in2 := 3)
      wire#w2
      Coil( "DB347_M_UNIT_1_STA_3".M_CODES_UNIT_1_STA_3.Ack_M903 )
   END_RUNG
   RUNG wire#w1
      I_Contact( "DB7253_UNIT_1_STA_3_MEAS_ENABLE_DISABLE".ENABLED )
   END_RUNG wire#w2
   RUNG wire#w1
      Contact( "DB2031_CYCLES_GENERAL".DRY_CYCLE.CYCLE_SELECTED )
   END_RUNG wire#w2
   RUNG wire#w1
      Contact( "DB2031_CYCLES_GENERAL".ROBOT_DRY_CYCLE.CYCLE_SELECTED )
   END_RUNG wire#w2
   // the same network as SCL:
   "DB347_M_UNIT_1_STA_3".M_CODES_UNIT_1_STA_3.Ack_M903 := "DB347_M_UNIT_1_STA_3".M_CODES_UNIT_1_STA_3.M903 AND (("DB16001_U1_STA3_MEAS_CLIENT_INTERFACE".U01_STA3_MEAS_Read.Variable.Status <> 3) OR NOT "DB7253_UNIT_1_STA_3_MEAS_ENABLE_DISABLE".ENABLED OR "DB2031_CYCLES_GENERAL".DRY_CYCLE.CYCLE_SELECTED OR "DB2031_CYCLES_GENERAL".ROBOT_DRY_CYCLE.CYCLE_SELECTED);
END_REGION

REGION Network 30: M903- STATION 3 MEASURMENT PC STOP LAYER THICKNESS MEASUREMENT
   RUNG wire#powerrail
      Contact( "DB332_EXTENDED_M_CODE_UNIT_1_STA_3".M_code[903] )
      wire#w1
      I_Contact( "DB347_M_UNIT_1_STA_3".M_CODES_UNIT_1_STA_3.Ack_M903 )
      I_Contact( "DB2120_MPP_ITC_IPC".RESET_FAULTS )
      I_Contact( "DB347_M_UNIT_1_STA_3".M_CODES_UNIT_1_STA_3.M_RESET_PULSE )
      Coil( "DB347_M_UNIT_1_STA_3".M_CODES_UNIT_1_STA_3.M903 )
   END_RUNG
   RUNG wire#powerrail
      Contact( "DB347_M_UNIT_1_STA_3".M_CODES_UNIT_1_STA_3.M903 )
   END_RUNG wire#w1
   // the same network as SCL:
   "DB347_M_UNIT_1_STA_3".M_CODES_UNIT_1_STA_3.M903 := ("DB332_EXTENDED_M_CODE_UNIT_1_STA_3".M_code[903] OR "DB347_M_UNIT_1_STA_3".M_CODES_UNIT_1_STA_3.M903) AND NOT "DB347_M_UNIT_1_STA_3".M_CODES_UNIT_1_STA_3.Ack_M903 AND NOT "DB2120_MPP_ITC_IPC".RESET_FAULTS AND NOT "DB347_M_UNIT_1_STA_3".M_CODES_UNIT_1_STA_3.M_RESET_PULSE;
END_REGION

REGION Network 31: ACKNOWLEDGE M904- STATION 3 MEASUREMENT PC START CALIBRATION
   RUNG wire#powerrail
      Contact( "DB347_M_UNIT_1_STA_3".M_CODES_UNIT_1_STA_3.M904 )
      wire#w1
      { S7_Templates := "SrcType := Int" } EQ_Contact(in1 := "DB16001_U1_STA3_MEAS_CLIENT_INTERFACE".U01_STA3_MEAS_Read.Variable.Status, in2 := 1)
      wire#w2
      Coil( "DB347_M_UNIT_1_STA_3".M_CODES_UNIT_1_STA_3.Ack_M904 )
   END_RUNG
   RUNG wire#w1
      I_Contact( "DB7253_UNIT_1_STA_3_MEAS_ENABLE_DISABLE".ENABLED )
   END_RUNG wire#w2
   RUNG wire#w1
      Contact( "DB2031_CYCLES_GENERAL".DRY_CYCLE.CYCLE_SELECTED )
   END_RUNG wire#w2
   RUNG wire#w1
      Contact( "DB2031_CYCLES_GENERAL".ROBOT_DRY_CYCLE.CYCLE_SELECTED )
   END_RUNG wire#w2
   // the same network as SCL:
   "DB347_M_UNIT_1_STA_3".M_CODES_UNIT_1_STA_3.Ack_M904 := "DB347_M_UNIT_1_STA_3".M_CODES_UNIT_1_STA_3.M904 AND (("DB16001_U1_STA3_MEAS_CLIENT_INTERFACE".U01_STA3_MEAS_Read.Variable.Status = 1) OR NOT "DB7253_UNIT_1_STA_3_MEAS_ENABLE_DISABLE".ENABLED OR "DB2031_CYCLES_GENERAL".DRY_CYCLE.CYCLE_SELECTED OR "DB2031_CYCLES_GENERAL".ROBOT_DRY_CYCLE.CYCLE_SELECTED);
END_REGION

REGION Network 32: M904- STATION 3 MEASUREMENT PC START CALIBRATION
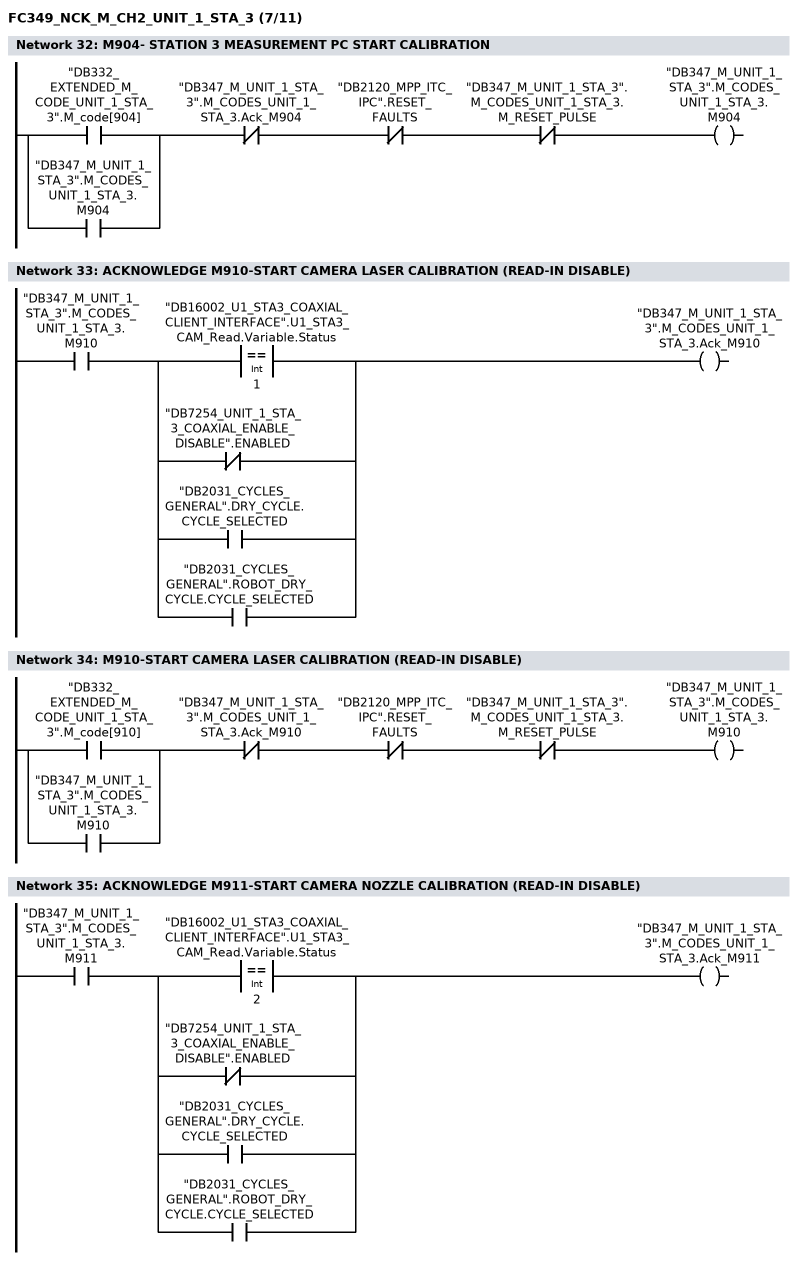
   RUNG wire#powerrail
      Contact( "DB332_EXTENDED_M_CODE_UNIT_1_STA_3".M_code[904] )
      wire#w1
      I_Contact( "DB347_M_UNIT_1_STA_3".M_CODES_UNIT_1_STA_3.Ack_M904 )
      I_Contact( "DB2120_MPP_ITC_IPC".RESET_FAULTS )
      I_Contact( "DB347_M_UNIT_1_STA_3".M_CODES_UNIT_1_STA_3.M_RESET_PULSE )
      Coil( "DB347_M_UNIT_1_STA_3".M_CODES_UNIT_1_STA_3.M904 )
   END_RUNG
   RUNG wire#powerrail
      Contact( "DB347_M_UNIT_1_STA_3".M_CODES_UNIT_1_STA_3.M904 )
   END_RUNG wire#w1
   // the same network as SCL:
   "DB347_M_UNIT_1_STA_3".M_CODES_UNIT_1_STA_3.M904 := ("DB332_EXTENDED_M_CODE_UNIT_1_STA_3".M_code[904] OR "DB347_M_UNIT_1_STA_3".M_CODES_UNIT_1_STA_3.M904) AND NOT "DB347_M_UNIT_1_STA_3".M_CODES_UNIT_1_STA_3.Ack_M904 AND NOT "DB2120_MPP_ITC_IPC".RESET_FAULTS AND NOT "DB347_M_UNIT_1_STA_3".M_CODES_UNIT_1_STA_3.M_RESET_PULSE;
END_REGION

REGION Network 33: ACKNOWLEDGE M910-START CAMERA LASER CALIBRATION (READ-IN DISABLE)
   RUNG wire#powerrail
      Contact( "DB347_M_UNIT_1_STA_3".M_CODES_UNIT_1_STA_3.M910 )
      wire#w1
      { S7_Templates := "SrcType := Int" } EQ_Contact(in1 := "DB16002_U1_STA3_COAXIAL_CLIENT_INTERFACE".U1_STA3_CAM_Read.Variable.Status, in2 := 1)
      wire#w2
      Coil( "DB347_M_UNIT_1_STA_3".M_CODES_UNIT_1_STA_3.Ack_M910 )
   END_RUNG
   RUNG wire#w1
      I_Contact( "DB7254_UNIT_1_STA_3_COAXIAL_ENABLE_DISABLE".ENABLED )
   END_RUNG wire#w2
   RUNG wire#w1
      Contact( "DB2031_CYCLES_GENERAL".DRY_CYCLE.CYCLE_SELECTED )
   END_RUNG wire#w2
   RUNG wire#w1
      Contact( "DB2031_CYCLES_GENERAL".ROBOT_DRY_CYCLE.CYCLE_SELECTED )
   END_RUNG wire#w2
   // the same network as SCL:
   "DB347_M_UNIT_1_STA_3".M_CODES_UNIT_1_STA_3.Ack_M910 := "DB347_M_UNIT_1_STA_3".M_CODES_UNIT_1_STA_3.M910 AND (("DB16002_U1_STA3_COAXIAL_CLIENT_INTERFACE".U1_STA3_CAM_Read.Variable.Status = 1) OR NOT "DB7254_UNIT_1_STA_3_COAXIAL_ENABLE_DISABLE".ENABLED OR "DB2031_CYCLES_GENERAL".DRY_CYCLE.CYCLE_SELECTED OR "DB2031_CYCLES_GENERAL".ROBOT_DRY_CYCLE.CYCLE_SELECTED);
END_REGION

REGION Network 34: M910-START CAMERA LASER CALIBRATION (READ-IN DISABLE)
   RUNG wire#powerrail
      Contact( "DB332_EXTENDED_M_CODE_UNIT_1_STA_3".M_code[910] )
      wire#w1
      I_Contact( "DB347_M_UNIT_1_STA_3".M_CODES_UNIT_1_STA_3.Ack_M910 )
      I_Contact( "DB2120_MPP_ITC_IPC".RESET_FAULTS )
      I_Contact( "DB347_M_UNIT_1_STA_3".M_CODES_UNIT_1_STA_3.M_RESET_PULSE )
      Coil( "DB347_M_UNIT_1_STA_3".M_CODES_UNIT_1_STA_3.M910 )
   END_RUNG
   RUNG wire#powerrail
      Contact( "DB347_M_UNIT_1_STA_3".M_CODES_UNIT_1_STA_3.M910 )
   END_RUNG wire#w1
   // the same network as SCL:
   "DB347_M_UNIT_1_STA_3".M_CODES_UNIT_1_STA_3.M910 := ("DB332_EXTENDED_M_CODE_UNIT_1_STA_3".M_code[910] OR "DB347_M_UNIT_1_STA_3".M_CODES_UNIT_1_STA_3.M910) AND NOT "DB347_M_UNIT_1_STA_3".M_CODES_UNIT_1_STA_3.Ack_M910 AND NOT "DB2120_MPP_ITC_IPC".RESET_FAULTS AND NOT "DB347_M_UNIT_1_STA_3".M_CODES_UNIT_1_STA_3.M_RESET_PULSE;
END_REGION

REGION Network 35: ACKNOWLEDGE M911-START CAMERA NOZZLE CALIBRATION (READ-IN DISABLE)
   RUNG wire#powerrail
      Contact( "DB347_M_UNIT_1_STA_3".M_CODES_UNIT_1_STA_3.M911 )
      wire#w1
      { S7_Templates := "SrcType := Int" } EQ_Contact(in1 := "DB16002_U1_STA3_COAXIAL_CLIENT_INTERFACE".U1_STA3_CAM_Read.Variable.Status, in2 := 2)
      wire#w2
      Coil( "DB347_M_UNIT_1_STA_3".M_CODES_UNIT_1_STA_3.Ack_M911 )
   END_RUNG
   RUNG wire#w1
      I_Contact( "DB7254_UNIT_1_STA_3_COAXIAL_ENABLE_DISABLE".ENABLED )
   END_RUNG wire#w2
   RUNG wire#w1
      Contact( "DB2031_CYCLES_GENERAL".DRY_CYCLE.CYCLE_SELECTED )
   END_RUNG wire#w2
   RUNG wire#w1
      Contact( "DB2031_CYCLES_GENERAL".ROBOT_DRY_CYCLE.CYCLE_SELECTED )
   END_RUNG wire#w2
   // the same network as SCL:
   "DB347_M_UNIT_1_STA_3".M_CODES_UNIT_1_STA_3.Ack_M911 := "DB347_M_UNIT_1_STA_3".M_CODES_UNIT_1_STA_3.M911 AND (("DB16002_U1_STA3_COAXIAL_CLIENT_INTERFACE".U1_STA3_CAM_Read.Variable.Status = 2) OR NOT "DB7254_UNIT_1_STA_3_COAXIAL_ENABLE_DISABLE".ENABLED OR "DB2031_CYCLES_GENERAL".DRY_CYCLE.CYCLE_SELECTED OR "DB2031_CYCLES_GENERAL".ROBOT_DRY_CYCLE.CYCLE_SELECTED);
END_REGION

REGION Network 36: M911-START CAMERA NOZZLE CALIBRATION (READ-IN DISABLE)
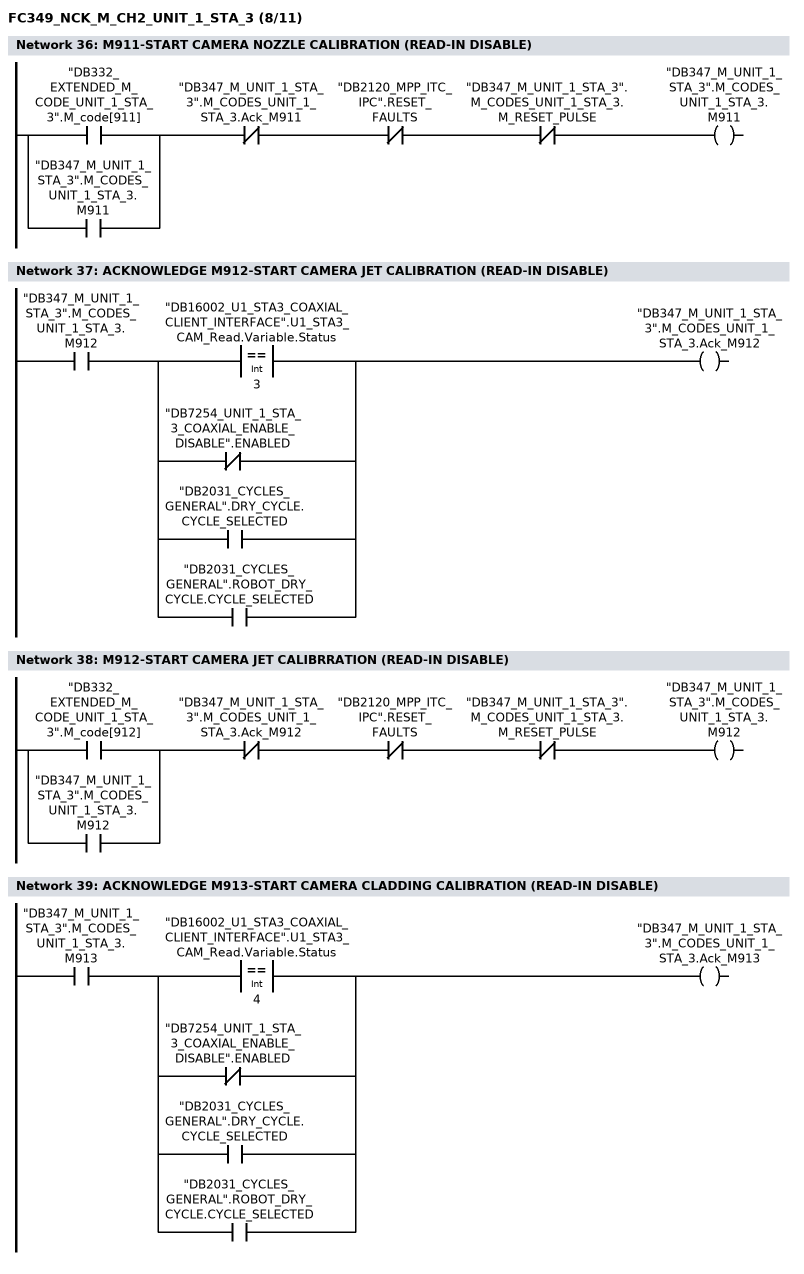
   RUNG wire#powerrail
      Contact( "DB332_EXTENDED_M_CODE_UNIT_1_STA_3".M_code[911] )
      wire#w1
      I_Contact( "DB347_M_UNIT_1_STA_3".M_CODES_UNIT_1_STA_3.Ack_M911 )
      I_Contact( "DB2120_MPP_ITC_IPC".RESET_FAULTS )
      I_Contact( "DB347_M_UNIT_1_STA_3".M_CODES_UNIT_1_STA_3.M_RESET_PULSE )
      Coil( "DB347_M_UNIT_1_STA_3".M_CODES_UNIT_1_STA_3.M911 )
   END_RUNG
   RUNG wire#powerrail
      Contact( "DB347_M_UNIT_1_STA_3".M_CODES_UNIT_1_STA_3.M911 )
   END_RUNG wire#w1
   // the same network as SCL:
   "DB347_M_UNIT_1_STA_3".M_CODES_UNIT_1_STA_3.M911 := ("DB332_EXTENDED_M_CODE_UNIT_1_STA_3".M_code[911] OR "DB347_M_UNIT_1_STA_3".M_CODES_UNIT_1_STA_3.M911) AND NOT "DB347_M_UNIT_1_STA_3".M_CODES_UNIT_1_STA_3.Ack_M911 AND NOT "DB2120_MPP_ITC_IPC".RESET_FAULTS AND NOT "DB347_M_UNIT_1_STA_3".M_CODES_UNIT_1_STA_3.M_RESET_PULSE;
END_REGION

REGION Network 37: ACKNOWLEDGE M912-START CAMERA JET CALIBRATION (READ-IN DISABLE)
   RUNG wire#powerrail
      Contact( "DB347_M_UNIT_1_STA_3".M_CODES_UNIT_1_STA_3.M912 )
      wire#w1
      { S7_Templates := "SrcType := Int" } EQ_Contact(in1 := "DB16002_U1_STA3_COAXIAL_CLIENT_INTERFACE".U1_STA3_CAM_Read.Variable.Status, in2 := 3)
      wire#w2
      Coil( "DB347_M_UNIT_1_STA_3".M_CODES_UNIT_1_STA_3.Ack_M912 )
   END_RUNG
   RUNG wire#w1
      I_Contact( "DB7254_UNIT_1_STA_3_COAXIAL_ENABLE_DISABLE".ENABLED )
   END_RUNG wire#w2
   RUNG wire#w1
      Contact( "DB2031_CYCLES_GENERAL".DRY_CYCLE.CYCLE_SELECTED )
   END_RUNG wire#w2
   RUNG wire#w1
      Contact( "DB2031_CYCLES_GENERAL".ROBOT_DRY_CYCLE.CYCLE_SELECTED )
   END_RUNG wire#w2
   // the same network as SCL:
   "DB347_M_UNIT_1_STA_3".M_CODES_UNIT_1_STA_3.Ack_M912 := "DB347_M_UNIT_1_STA_3".M_CODES_UNIT_1_STA_3.M912 AND (("DB16002_U1_STA3_COAXIAL_CLIENT_INTERFACE".U1_STA3_CAM_Read.Variable.Status = 3) OR NOT "DB7254_UNIT_1_STA_3_COAXIAL_ENABLE_DISABLE".ENABLED OR "DB2031_CYCLES_GENERAL".DRY_CYCLE.CYCLE_SELECTED OR "DB2031_CYCLES_GENERAL".ROBOT_DRY_CYCLE.CYCLE_SELECTED);
END_REGION

REGION Network 38: M912-START CAMERA JET CALIBRRATION (READ-IN DISABLE)
   RUNG wire#powerrail
      Contact( "DB332_EXTENDED_M_CODE_UNIT_1_STA_3".M_code[912] )
      wire#w1
      I_Contact( "DB347_M_UNIT_1_STA_3".M_CODES_UNIT_1_STA_3.Ack_M912 )
      I_Contact( "DB2120_MPP_ITC_IPC".RESET_FAULTS )
      I_Contact( "DB347_M_UNIT_1_STA_3".M_CODES_UNIT_1_STA_3.M_RESET_PULSE )
      Coil( "DB347_M_UNIT_1_STA_3".M_CODES_UNIT_1_STA_3.M912 )
   END_RUNG
   RUNG wire#powerrail
      Contact( "DB347_M_UNIT_1_STA_3".M_CODES_UNIT_1_STA_3.M912 )
   END_RUNG wire#w1
   // the same network as SCL:
   "DB347_M_UNIT_1_STA_3".M_CODES_UNIT_1_STA_3.M912 := ("DB332_EXTENDED_M_CODE_UNIT_1_STA_3".M_code[912] OR "DB347_M_UNIT_1_STA_3".M_CODES_UNIT_1_STA_3.M912) AND NOT "DB347_M_UNIT_1_STA_3".M_CODES_UNIT_1_STA_3.Ack_M912 AND NOT "DB2120_MPP_ITC_IPC".RESET_FAULTS AND NOT "DB347_M_UNIT_1_STA_3".M_CODES_UNIT_1_STA_3.M_RESET_PULSE;
END_REGION

REGION Network 39: ACKNOWLEDGE M913-START CAMERA CLADDING CALIBRATION (READ-IN DISABLE)
   RUNG wire#powerrail
      Contact( "DB347_M_UNIT_1_STA_3".M_CODES_UNIT_1_STA_3.M913 )
      wire#w1
      { S7_Templates := "SrcType := Int" } EQ_Contact(in1 := "DB16002_U1_STA3_COAXIAL_CLIENT_INTERFACE".U1_STA3_CAM_Read.Variable.Status, in2 := 4)
      wire#w2
      Coil( "DB347_M_UNIT_1_STA_3".M_CODES_UNIT_1_STA_3.Ack_M913 )
   END_RUNG
   RUNG wire#w1
      I_Contact( "DB7254_UNIT_1_STA_3_COAXIAL_ENABLE_DISABLE".ENABLED )
   END_RUNG wire#w2
   RUNG wire#w1
      Contact( "DB2031_CYCLES_GENERAL".DRY_CYCLE.CYCLE_SELECTED )
   END_RUNG wire#w2
   RUNG wire#w1
      Contact( "DB2031_CYCLES_GENERAL".ROBOT_DRY_CYCLE.CYCLE_SELECTED )
   END_RUNG wire#w2
   // the same network as SCL:
   "DB347_M_UNIT_1_STA_3".M_CODES_UNIT_1_STA_3.Ack_M913 := "DB347_M_UNIT_1_STA_3".M_CODES_UNIT_1_STA_3.M913 AND (("DB16002_U1_STA3_COAXIAL_CLIENT_INTERFACE".U1_STA3_CAM_Read.Variable.Status = 4) OR NOT "DB7254_UNIT_1_STA_3_COAXIAL_ENABLE_DISABLE".ENABLED OR "DB2031_CYCLES_GENERAL".DRY_CYCLE.CYCLE_SELECTED OR "DB2031_CYCLES_GENERAL".ROBOT_DRY_CYCLE.CYCLE_SELECTED);
END_REGION

REGION Network 40: M913-START CAMERA CLADDING CALIBRATION (READ-IN DISABLE)
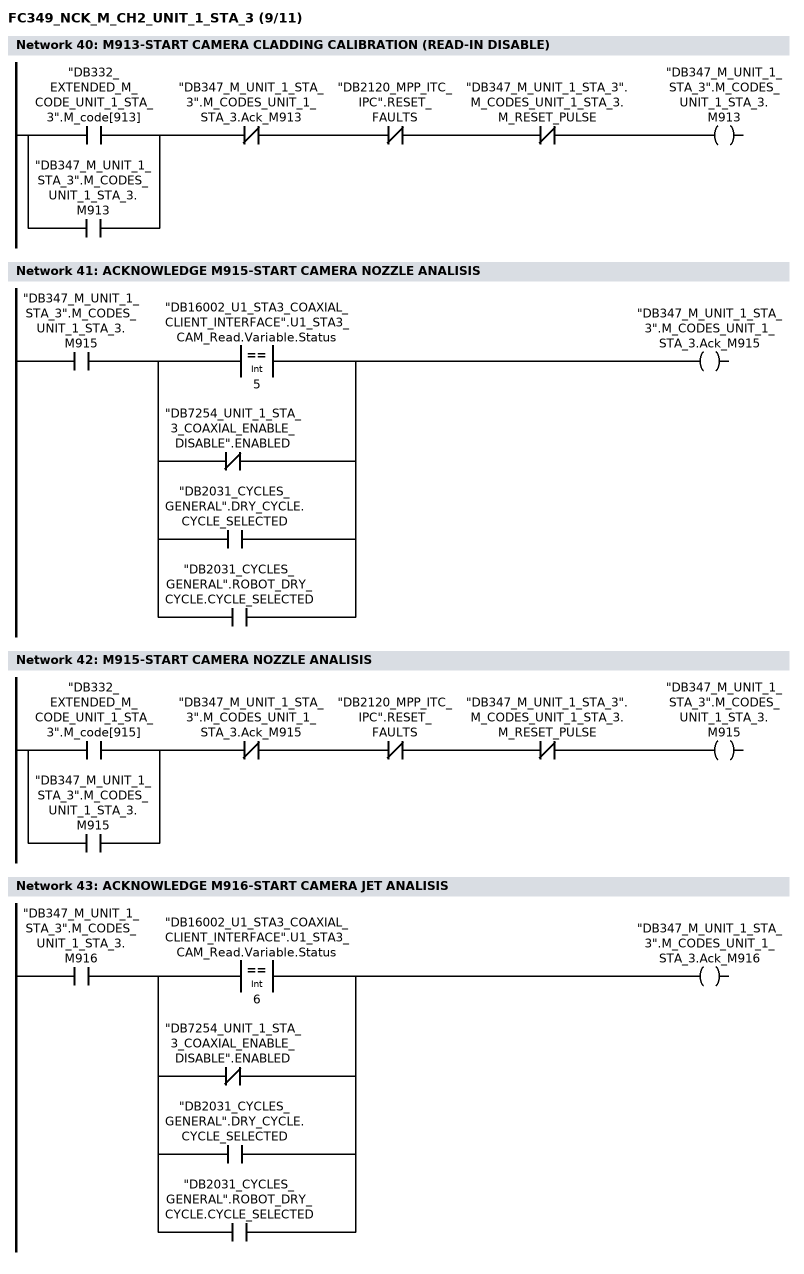
   RUNG wire#powerrail
      Contact( "DB332_EXTENDED_M_CODE_UNIT_1_STA_3".M_code[913] )
      wire#w1
      I_Contact( "DB347_M_UNIT_1_STA_3".M_CODES_UNIT_1_STA_3.Ack_M913 )
      I_Contact( "DB2120_MPP_ITC_IPC".RESET_FAULTS )
      I_Contact( "DB347_M_UNIT_1_STA_3".M_CODES_UNIT_1_STA_3.M_RESET_PULSE )
      Coil( "DB347_M_UNIT_1_STA_3".M_CODES_UNIT_1_STA_3.M913 )
   END_RUNG
   RUNG wire#powerrail
      Contact( "DB347_M_UNIT_1_STA_3".M_CODES_UNIT_1_STA_3.M913 )
   END_RUNG wire#w1
   // the same network as SCL:
   "DB347_M_UNIT_1_STA_3".M_CODES_UNIT_1_STA_3.M913 := ("DB332_EXTENDED_M_CODE_UNIT_1_STA_3".M_code[913] OR "DB347_M_UNIT_1_STA_3".M_CODES_UNIT_1_STA_3.M913) AND NOT "DB347_M_UNIT_1_STA_3".M_CODES_UNIT_1_STA_3.Ack_M913 AND NOT "DB2120_MPP_ITC_IPC".RESET_FAULTS AND NOT "DB347_M_UNIT_1_STA_3".M_CODES_UNIT_1_STA_3.M_RESET_PULSE;
END_REGION

REGION Network 41: ACKNOWLEDGE M915-START CAMERA NOZZLE ANALISIS
   RUNG wire#powerrail
      Contact( "DB347_M_UNIT_1_STA_3".M_CODES_UNIT_1_STA_3.M915 )
      wire#w1
      { S7_Templates := "SrcType := Int" } EQ_Contact(in1 := "DB16002_U1_STA3_COAXIAL_CLIENT_INTERFACE".U1_STA3_CAM_Read.Variable.Status, in2 := 5)
      wire#w2
      Coil( "DB347_M_UNIT_1_STA_3".M_CODES_UNIT_1_STA_3.Ack_M915 )
   END_RUNG
   RUNG wire#w1
      I_Contact( "DB7254_UNIT_1_STA_3_COAXIAL_ENABLE_DISABLE".ENABLED )
   END_RUNG wire#w2
   RUNG wire#w1
      Contact( "DB2031_CYCLES_GENERAL".DRY_CYCLE.CYCLE_SELECTED )
   END_RUNG wire#w2
   RUNG wire#w1
      Contact( "DB2031_CYCLES_GENERAL".ROBOT_DRY_CYCLE.CYCLE_SELECTED )
   END_RUNG wire#w2
   // the same network as SCL:
   "DB347_M_UNIT_1_STA_3".M_CODES_UNIT_1_STA_3.Ack_M915 := "DB347_M_UNIT_1_STA_3".M_CODES_UNIT_1_STA_3.M915 AND (("DB16002_U1_STA3_COAXIAL_CLIENT_INTERFACE".U1_STA3_CAM_Read.Variable.Status = 5) OR NOT "DB7254_UNIT_1_STA_3_COAXIAL_ENABLE_DISABLE".ENABLED OR "DB2031_CYCLES_GENERAL".DRY_CYCLE.CYCLE_SELECTED OR "DB2031_CYCLES_GENERAL".ROBOT_DRY_CYCLE.CYCLE_SELECTED);
END_REGION

REGION Network 42: M915-START CAMERA NOZZLE ANALISIS
   RUNG wire#powerrail
      Contact( "DB332_EXTENDED_M_CODE_UNIT_1_STA_3".M_code[915] )
      wire#w1
      I_Contact( "DB347_M_UNIT_1_STA_3".M_CODES_UNIT_1_STA_3.Ack_M915 )
      I_Contact( "DB2120_MPP_ITC_IPC".RESET_FAULTS )
      I_Contact( "DB347_M_UNIT_1_STA_3".M_CODES_UNIT_1_STA_3.M_RESET_PULSE )
      Coil( "DB347_M_UNIT_1_STA_3".M_CODES_UNIT_1_STA_3.M915 )
   END_RUNG
   RUNG wire#powerrail
      Contact( "DB347_M_UNIT_1_STA_3".M_CODES_UNIT_1_STA_3.M915 )
   END_RUNG wire#w1
   // the same network as SCL:
   "DB347_M_UNIT_1_STA_3".M_CODES_UNIT_1_STA_3.M915 := ("DB332_EXTENDED_M_CODE_UNIT_1_STA_3".M_code[915] OR "DB347_M_UNIT_1_STA_3".M_CODES_UNIT_1_STA_3.M915) AND NOT "DB347_M_UNIT_1_STA_3".M_CODES_UNIT_1_STA_3.Ack_M915 AND NOT "DB2120_MPP_ITC_IPC".RESET_FAULTS AND NOT "DB347_M_UNIT_1_STA_3".M_CODES_UNIT_1_STA_3.M_RESET_PULSE;
END_REGION

REGION Network 43: ACKNOWLEDGE M916-START CAMERA JET ANALISIS
   RUNG wire#powerrail
      Contact( "DB347_M_UNIT_1_STA_3".M_CODES_UNIT_1_STA_3.M916 )
      wire#w1
      { S7_Templates := "SrcType := Int" } EQ_Contact(in1 := "DB16002_U1_STA3_COAXIAL_CLIENT_INTERFACE".U1_STA3_CAM_Read.Variable.Status, in2 := 6)
      wire#w2
      Coil( "DB347_M_UNIT_1_STA_3".M_CODES_UNIT_1_STA_3.Ack_M916 )
   END_RUNG
   RUNG wire#w1
      I_Contact( "DB7254_UNIT_1_STA_3_COAXIAL_ENABLE_DISABLE".ENABLED )
   END_RUNG wire#w2
   RUNG wire#w1
      Contact( "DB2031_CYCLES_GENERAL".DRY_CYCLE.CYCLE_SELECTED )
   END_RUNG wire#w2
   RUNG wire#w1
      Contact( "DB2031_CYCLES_GENERAL".ROBOT_DRY_CYCLE.CYCLE_SELECTED )
   END_RUNG wire#w2
   // the same network as SCL:
   "DB347_M_UNIT_1_STA_3".M_CODES_UNIT_1_STA_3.Ack_M916 := "DB347_M_UNIT_1_STA_3".M_CODES_UNIT_1_STA_3.M916 AND (("DB16002_U1_STA3_COAXIAL_CLIENT_INTERFACE".U1_STA3_CAM_Read.Variable.Status = 6) OR NOT "DB7254_UNIT_1_STA_3_COAXIAL_ENABLE_DISABLE".ENABLED OR "DB2031_CYCLES_GENERAL".DRY_CYCLE.CYCLE_SELECTED OR "DB2031_CYCLES_GENERAL".ROBOT_DRY_CYCLE.CYCLE_SELECTED);
END_REGION

REGION Network 44: M916-START CAMERA JET ANALISIS
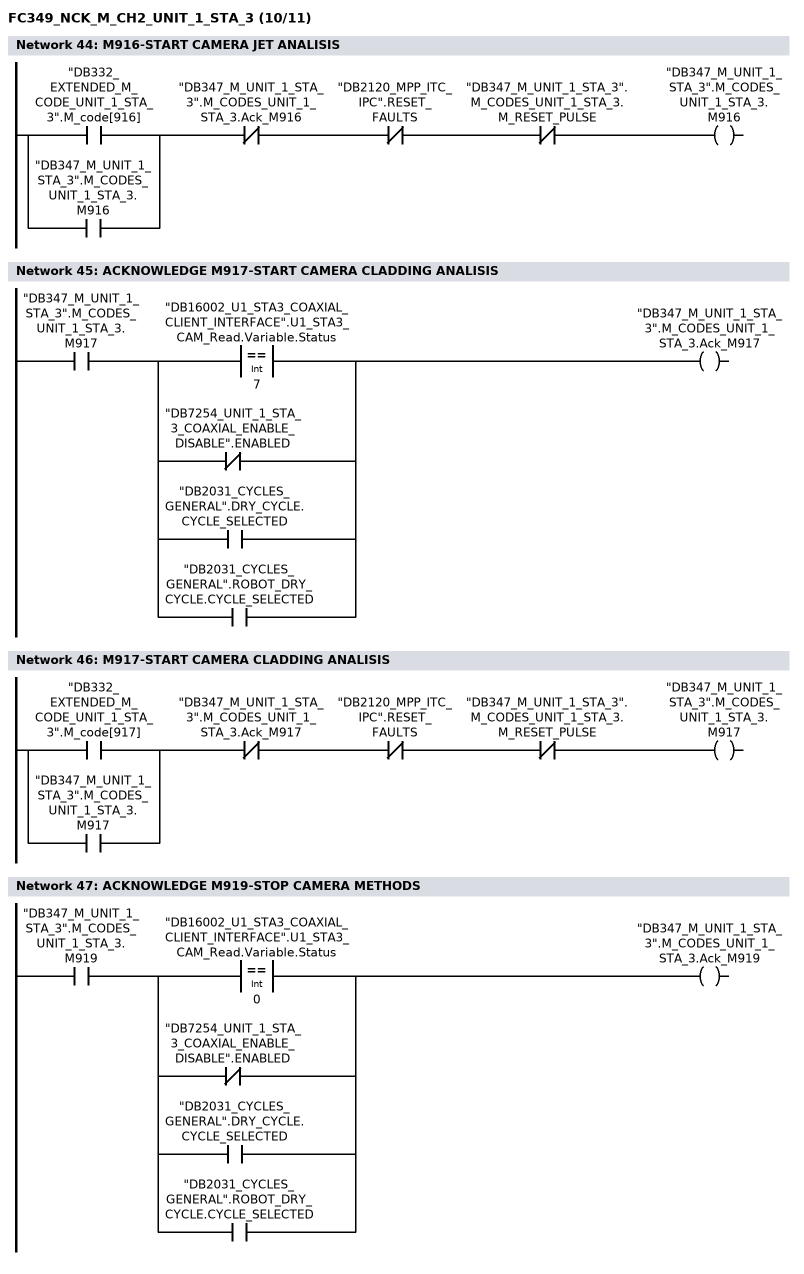
   RUNG wire#powerrail
      Contact( "DB332_EXTENDED_M_CODE_UNIT_1_STA_3".M_code[916] )
      wire#w1
      I_Contact( "DB347_M_UNIT_1_STA_3".M_CODES_UNIT_1_STA_3.Ack_M916 )
      I_Contact( "DB2120_MPP_ITC_IPC".RESET_FAULTS )
      I_Contact( "DB347_M_UNIT_1_STA_3".M_CODES_UNIT_1_STA_3.M_RESET_PULSE )
      Coil( "DB347_M_UNIT_1_STA_3".M_CODES_UNIT_1_STA_3.M916 )
   END_RUNG
   RUNG wire#powerrail
      Contact( "DB347_M_UNIT_1_STA_3".M_CODES_UNIT_1_STA_3.M916 )
   END_RUNG wire#w1
   // the same network as SCL:
   "DB347_M_UNIT_1_STA_3".M_CODES_UNIT_1_STA_3.M916 := ("DB332_EXTENDED_M_CODE_UNIT_1_STA_3".M_code[916] OR "DB347_M_UNIT_1_STA_3".M_CODES_UNIT_1_STA_3.M916) AND NOT "DB347_M_UNIT_1_STA_3".M_CODES_UNIT_1_STA_3.Ack_M916 AND NOT "DB2120_MPP_ITC_IPC".RESET_FAULTS AND NOT "DB347_M_UNIT_1_STA_3".M_CODES_UNIT_1_STA_3.M_RESET_PULSE;
END_REGION

REGION Network 45: ACKNOWLEDGE M917-START CAMERA CLADDING ANALISIS
   RUNG wire#powerrail
      Contact( "DB347_M_UNIT_1_STA_3".M_CODES_UNIT_1_STA_3.M917 )
      wire#w1
      { S7_Templates := "SrcType := Int" } EQ_Contact(in1 := "DB16002_U1_STA3_COAXIAL_CLIENT_INTERFACE".U1_STA3_CAM_Read.Variable.Status, in2 := 7)
      wire#w2
      Coil( "DB347_M_UNIT_1_STA_3".M_CODES_UNIT_1_STA_3.Ack_M917 )
   END_RUNG
   RUNG wire#w1
      I_Contact( "DB7254_UNIT_1_STA_3_COAXIAL_ENABLE_DISABLE".ENABLED )
   END_RUNG wire#w2
   RUNG wire#w1
      Contact( "DB2031_CYCLES_GENERAL".DRY_CYCLE.CYCLE_SELECTED )
   END_RUNG wire#w2
   RUNG wire#w1
      Contact( "DB2031_CYCLES_GENERAL".ROBOT_DRY_CYCLE.CYCLE_SELECTED )
   END_RUNG wire#w2
   // the same network as SCL:
   "DB347_M_UNIT_1_STA_3".M_CODES_UNIT_1_STA_3.Ack_M917 := "DB347_M_UNIT_1_STA_3".M_CODES_UNIT_1_STA_3.M917 AND (("DB16002_U1_STA3_COAXIAL_CLIENT_INTERFACE".U1_STA3_CAM_Read.Variable.Status = 7) OR NOT "DB7254_UNIT_1_STA_3_COAXIAL_ENABLE_DISABLE".ENABLED OR "DB2031_CYCLES_GENERAL".DRY_CYCLE.CYCLE_SELECTED OR "DB2031_CYCLES_GENERAL".ROBOT_DRY_CYCLE.CYCLE_SELECTED);
END_REGION

REGION Network 46: M917-START CAMERA CLADDING ANALISIS
   RUNG wire#powerrail
      Contact( "DB332_EXTENDED_M_CODE_UNIT_1_STA_3".M_code[917] )
      wire#w1
      I_Contact( "DB347_M_UNIT_1_STA_3".M_CODES_UNIT_1_STA_3.Ack_M917 )
      I_Contact( "DB2120_MPP_ITC_IPC".RESET_FAULTS )
      I_Contact( "DB347_M_UNIT_1_STA_3".M_CODES_UNIT_1_STA_3.M_RESET_PULSE )
      Coil( "DB347_M_UNIT_1_STA_3".M_CODES_UNIT_1_STA_3.M917 )
   END_RUNG
   RUNG wire#powerrail
      Contact( "DB347_M_UNIT_1_STA_3".M_CODES_UNIT_1_STA_3.M917 )
   END_RUNG wire#w1
   // the same network as SCL:
   "DB347_M_UNIT_1_STA_3".M_CODES_UNIT_1_STA_3.M917 := ("DB332_EXTENDED_M_CODE_UNIT_1_STA_3".M_code[917] OR "DB347_M_UNIT_1_STA_3".M_CODES_UNIT_1_STA_3.M917) AND NOT "DB347_M_UNIT_1_STA_3".M_CODES_UNIT_1_STA_3.Ack_M917 AND NOT "DB2120_MPP_ITC_IPC".RESET_FAULTS AND NOT "DB347_M_UNIT_1_STA_3".M_CODES_UNIT_1_STA_3.M_RESET_PULSE;
END_REGION

REGION Network 47: ACKNOWLEDGE M919-STOP CAMERA METHODS
   RUNG wire#powerrail
      Contact( "DB347_M_UNIT_1_STA_3".M_CODES_UNIT_1_STA_3.M919 )
      wire#w1
      { S7_Templates := "SrcType := Int" } EQ_Contact(in1 := "DB16002_U1_STA3_COAXIAL_CLIENT_INTERFACE".U1_STA3_CAM_Read.Variable.Status, in2 := 0)
      wire#w2
      Coil( "DB347_M_UNIT_1_STA_3".M_CODES_UNIT_1_STA_3.Ack_M919 )
   END_RUNG
   RUNG wire#w1
      I_Contact( "DB7254_UNIT_1_STA_3_COAXIAL_ENABLE_DISABLE".ENABLED )
   END_RUNG wire#w2
   RUNG wire#w1
      Contact( "DB2031_CYCLES_GENERAL".DRY_CYCLE.CYCLE_SELECTED )
   END_RUNG wire#w2
   RUNG wire#w1
      Contact( "DB2031_CYCLES_GENERAL".ROBOT_DRY_CYCLE.CYCLE_SELECTED )
   END_RUNG wire#w2
   // the same network as SCL:
   "DB347_M_UNIT_1_STA_3".M_CODES_UNIT_1_STA_3.Ack_M919 := "DB347_M_UNIT_1_STA_3".M_CODES_UNIT_1_STA_3.M919 AND (("DB16002_U1_STA3_COAXIAL_CLIENT_INTERFACE".U1_STA3_CAM_Read.Variable.Status = 0) OR NOT "DB7254_UNIT_1_STA_3_COAXIAL_ENABLE_DISABLE".ENABLED OR "DB2031_CYCLES_GENERAL".DRY_CYCLE.CYCLE_SELECTED OR "DB2031_CYCLES_GENERAL".ROBOT_DRY_CYCLE.CYCLE_SELECTED);
END_REGION

REGION Network 48: M919-STOP CAMERA METHODS
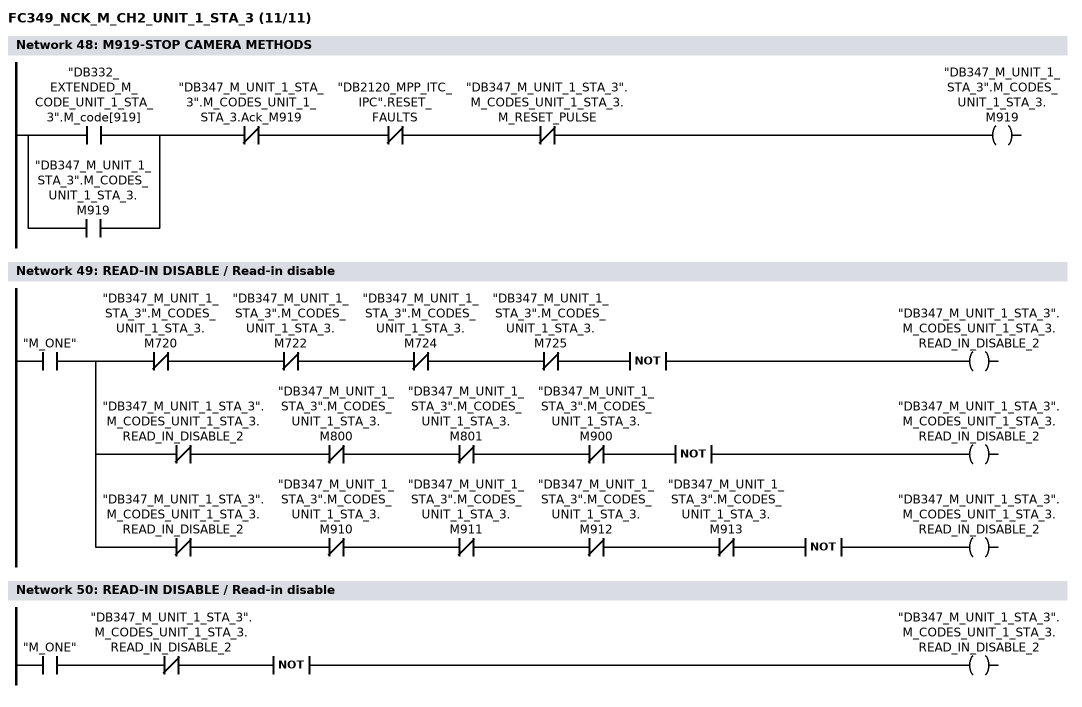
   RUNG wire#powerrail
      Contact( "DB332_EXTENDED_M_CODE_UNIT_1_STA_3".M_code[919] )
      wire#w1
      I_Contact( "DB347_M_UNIT_1_STA_3".M_CODES_UNIT_1_STA_3.Ack_M919 )
      I_Contact( "DB2120_MPP_ITC_IPC".RESET_FAULTS )
      I_Contact( "DB347_M_UNIT_1_STA_3".M_CODES_UNIT_1_STA_3.M_RESET_PULSE )
      Coil( "DB347_M_UNIT_1_STA_3".M_CODES_UNIT_1_STA_3.M919 )
   END_RUNG
   RUNG wire#powerrail
      Contact( "DB347_M_UNIT_1_STA_3".M_CODES_UNIT_1_STA_3.M919 )
   END_RUNG wire#w1
   // the same network as SCL:
   "DB347_M_UNIT_1_STA_3".M_CODES_UNIT_1_STA_3.M919 := ("DB332_EXTENDED_M_CODE_UNIT_1_STA_3".M_code[919] OR "DB347_M_UNIT_1_STA_3".M_CODES_UNIT_1_STA_3.M919) AND NOT "DB347_M_UNIT_1_STA_3".M_CODES_UNIT_1_STA_3.Ack_M919 AND NOT "DB2120_MPP_ITC_IPC".RESET_FAULTS AND NOT "DB347_M_UNIT_1_STA_3".M_CODES_UNIT_1_STA_3.M_RESET_PULSE;
END_REGION

REGION Network 49: READ-IN DISABLE / Read-in disable
   RUNG wire#powerrail
      Contact( "M_ONE" )
      wire#w1
      I_Contact( "DB347_M_UNIT_1_STA_3".M_CODES_UNIT_1_STA_3.M720 )
      I_Contact( "DB347_M_UNIT_1_STA_3".M_CODES_UNIT_1_STA_3.M722 )
      I_Contact( "DB347_M_UNIT_1_STA_3".M_CODES_UNIT_1_STA_3.M724 )
      I_Contact( "DB347_M_UNIT_1_STA_3".M_CODES_UNIT_1_STA_3.M725 )
      Not()
      Coil( "DB347_M_UNIT_1_STA_3".M_CODES_UNIT_1_STA_3.READ_IN_DISABLE_2 )
   END_RUNG
   RUNG wire#w1
      I_Contact( "DB347_M_UNIT_1_STA_3".M_CODES_UNIT_1_STA_3.READ_IN_DISABLE_2 )
      I_Contact( "DB347_M_UNIT_1_STA_3".M_CODES_UNIT_1_STA_3.M800 )
      I_Contact( "DB347_M_UNIT_1_STA_3".M_CODES_UNIT_1_STA_3.M801 )
      I_Contact( "DB347_M_UNIT_1_STA_3".M_CODES_UNIT_1_STA_3.M900 )
      Not()
      Coil( "DB347_M_UNIT_1_STA_3".M_CODES_UNIT_1_STA_3.READ_IN_DISABLE_2 )
   END_RUNG
   RUNG wire#w1
      I_Contact( "DB347_M_UNIT_1_STA_3".M_CODES_UNIT_1_STA_3.READ_IN_DISABLE_2 )
      I_Contact( "DB347_M_UNIT_1_STA_3".M_CODES_UNIT_1_STA_3.M910 )
      I_Contact( "DB347_M_UNIT_1_STA_3".M_CODES_UNIT_1_STA_3.M911 )
      I_Contact( "DB347_M_UNIT_1_STA_3".M_CODES_UNIT_1_STA_3.M912 )
      I_Contact( "DB347_M_UNIT_1_STA_3".M_CODES_UNIT_1_STA_3.M913 )
      Not()
      Coil( "DB347_M_UNIT_1_STA_3".M_CODES_UNIT_1_STA_3.READ_IN_DISABLE_2 )
   END_RUNG
   // the same network as SCL:
   "DB347_M_UNIT_1_STA_3".M_CODES_UNIT_1_STA_3.READ_IN_DISABLE_2 := NOT ("M_ONE" AND NOT "DB347_M_UNIT_1_STA_3".M_CODES_UNIT_1_STA_3.M720 AND NOT "DB347_M_UNIT_1_STA_3".M_CODES_UNIT_1_STA_3.M722 AND NOT "DB347_M_UNIT_1_STA_3".M_CODES_UNIT_1_STA_3.M724 AND NOT "DB347_M_UNIT_1_STA_3".M_CODES_UNIT_1_STA_3.M725);
   "DB347_M_UNIT_1_STA_3".M_CODES_UNIT_1_STA_3.READ_IN_DISABLE_2 := NOT ("M_ONE" AND NOT "DB347_M_UNIT_1_STA_3".M_CODES_UNIT_1_STA_3.READ_IN_DISABLE_2 AND NOT "DB347_M_UNIT_1_STA_3".M_CODES_UNIT_1_STA_3.M800 AND NOT "DB347_M_UNIT_1_STA_3".M_CODES_UNIT_1_STA_3.M801 AND NOT "DB347_M_UNIT_1_STA_3".M_CODES_UNIT_1_STA_3.M900);
   "DB347_M_UNIT_1_STA_3".M_CODES_UNIT_1_STA_3.READ_IN_DISABLE_2 := NOT ("M_ONE" AND NOT "DB347_M_UNIT_1_STA_3".M_CODES_UNIT_1_STA_3.READ_IN_DISABLE_2 AND NOT "DB347_M_UNIT_1_STA_3".M_CODES_UNIT_1_STA_3.M910 AND NOT "DB347_M_UNIT_1_STA_3".M_CODES_UNIT_1_STA_3.M911 AND NOT "DB347_M_UNIT_1_STA_3".M_CODES_UNIT_1_STA_3.M912 AND NOT "DB347_M_UNIT_1_STA_3".M_CODES_UNIT_1_STA_3.M913);
END_REGION

REGION Network 50: READ-IN DISABLE / Read-in disable
   RUNG wire#powerrail
      Contact( "M_ONE" )
      I_Contact( "DB347_M_UNIT_1_STA_3".M_CODES_UNIT_1_STA_3.READ_IN_DISABLE_2 )
      Not()
      Coil( "DB347_M_UNIT_1_STA_3".M_CODES_UNIT_1_STA_3.READ_IN_DISABLE_2 )
   END_RUNG
   // the same network as SCL:
   "DB347_M_UNIT_1_STA_3".M_CODES_UNIT_1_STA_3.READ_IN_DISABLE_2 := NOT ("M_ONE" AND NOT "DB347_M_UNIT_1_STA_3".M_CODES_UNIT_1_STA_3.READ_IN_DISABLE_2);
END_REGION
END_FUNCTION
